// TIA Portal V16 program export: 1 tag tables, 6 data types, 52 data blocks, 60 code blocks (in call order from the OBs), 9 instance data blocks

VAR_GLOBAL   // PLC tag table "Default tag table"
   "E0.4" AT %I0.4 : Bool;   // CONTROLLO SALDATORE FILM
   "E0.5" AT %I0.5 : Bool;   // RICHIESTA APERTURA PORTA
   "E0.6" AT %I0.6 : Bool;   // PRESSOSTATO MACCHINA
   "E0.7" AT %I0.7 : Bool;   // ALLARME TERMICO MACCHINA
   "E1.0" AT %I1.0 : Bool;   // EMERGENZA MACCHINA
   "E1.1" AT %I1.1 : Bool;   // BARRIERE IMPEGNATE ENTRATA
   "E1.2" AT %I1.2 : Bool;   // BARRIERE IMPEGNATE USCITA
   "E1.3" AT %I1.3 : Bool;   // RESET MACCHINA
   "E1.4" AT %I1.4 : Bool;   // MARCIA AUTOMATICA MACCHINA
   "E1.5" AT %I1.5 : Bool;   // ARRESTO MACCHINA
   "E2.0" AT %I2.0 : Bool;   // TAVOLA IN FASE
   "E2.1" AT %I2.1 : Bool;   // [spare] COMANDO FRENO MOTORE ROTAZIONE
   "E2.2" AT %I2.2 : Bool;   // CARRELLO BASSO
   "E2.3" AT %I2.3 : Bool;   // CARRELLO ALTO
   "E2.4" AT %I2.4 : Bool;   // TAGLIO INDIETRO
   "E2.5" AT %I2.5 : Bool;   // TAGLIO AVANTI
   "E2.6" AT %I2.6 : Bool;   // CONTRASTO SALDATORE INDIETRO
   "E2.7" AT %I2.7 : Bool;   // CONTRASTO SALDATORE BASSO
   "E3.0" AT %I3.0 : Bool;   // RISERVA
   "E3.1" AT %I3.1 : Bool;   // RISERVA
   "E3.2" AT %I3.2 : Bool;   // LETTURA CENTRAGGIO PALLET TRASPORTO CENTRO MACCHINA
   "E3.3" AT %I3.3 : Bool;   // CONTEGGIO CENTRAGGIO PALLET TRASPORTO CENTRO MACCHINA
   "E3.4" AT %I3.4 : Bool;   // CONTROLLO ROTAZIONE TAVOLA IN ENTRATA E LETTURA LUNGHEZZA PALLET
   "E3.5" AT %I3.5 : Bool;   // CONTROLLO ROTAZIONE TAVOLA IN USCITA E FINE CICLO
   "E3.6" AT %I3.6 : Bool;   // SEGNALE PALLET PRONTO IN ENTRATA
   "E3.7" AT %I3.7 : Bool;   // SEGNALE PRONTO A RICEVERE IN USCITA
   "E4.0" AT %I4.0 : Bool;   // SEGNALE FINE TRASFERIMENTO PALLET IN USCITA
   "E4.1" AT %I4.1 : Bool;   // SEGNALE ESCLUSIONE FASCIATURA
   "E4.2" AT %I4.2 : Bool;   // POSIZIONAMENTO PALLET TRASPORTO POS. 01
   "E4.3" AT %I4.3 : Bool;   // POSIZIONAMENTO PALLET TRASPORTO POS. 02
   "E4.4" AT %I4.4 : Bool;   // POSIZIONAMENTO PALLET TRASPORTO POS. 03
   "E4.5" AT %I4.5 : Bool;   // POSIZIONAMENTO PALLET TRASPORTO POS. 04
   "E4.6" AT %I4.6 : Bool;   // POSIZIONAMENTO PALLET TRASPORTO POS. 05
   "E5.1" AT %I5.1 : Bool;   // POSIZIONAMENTO PALLET TRASPORTO POS. 08
   "E5.3" AT %I5.3 : Bool;   // [B2783] CONTROLLO 2 POSIZIONAMENTO POS. 05
   "E6.0" AT %I6.0 : Bool;   // CARRELLO BASSO (TOP)
   "E6.1" AT %I6.1 : Bool;   // CARRELLO ALTO (TOP)
   "E6.2" AT %I6.2 : Bool;   // LETTURA ALTEZZA PALLET (TOP)
   "E6.3" AT %I6.3 : Bool;   // PINZA CHIUSA BLOCCO FILM (TOP)
   "E6.4" AT %I6.4 : Bool;   // TAGLIO FILM AVANTI (TOP)
   "E6.5" AT %I6.5 : Bool;   // TAGLIO FILM INDIETRO (TOP)
   "E6.6" AT %I6.6 : Bool;   // ROTTURA ESAURIMENTO FILM (TOP)
   "E7.0" AT %I7.0 : Bool;   // CARRELLO INDIETRO (TOP)
   "E7.1" AT %I7.1 : Bool;   // CARRELLO AVANTI POSIZIONE TAGLIO (TOP)
   "E7.3" AT %I7.3 : Bool;   // PINZA CHIUSA TRAINO FILM (TOP)
   "E7.4" AT %I7.4 : Bool;   // SICUREZZA AVANZAMENTO (TOP)
   "E7.5" AT %I7.5 : Bool;   // SICUREZZA DISCESA (TOP) SX
   "E7.6" AT %I7.6 : Bool;   // SICUREZZA DISCESA (TOP) DX
   "E7.7" AT %I7.7 : Bool;   // SICUREZZA CONTROLLO SGANCIO FRENI SAL.-DISC. (TOP)
   HSC2Value AT %ID1004 : DInt;   // Counter value for HSC2
   HSC1Value AT %ID1000 : DInt;
   "E4.7" AT %I4.7 : Bool;   // POSIZIONAMENTO PALLET TRASPORTO POS. 06
   "E5.0" AT %I5.0 : Bool;   // POSIZIONAMENTO PALLET TRASPORTO POS. 07
   "E5.2" AT %I5.2 : Bool;   // [B2782] CONTROLLO 1 POSIZIONAMENTO POS. 05
   "E5.4" AT %I5.4 : Bool;   // SEGNALE PORTA TAGLIAFUOCO APERTA
   "E5.5" AT %I5.5 : Bool;   // SEGNALE CHIUSURA PORTA TAGLIAFUOCO
   "E5.6" AT %I5.6 : Bool;   // SelectorBypass
   "E5.7" AT %I5.7 : Bool;   // Free
   "E6.7" AT %I6.7 : Bool;   // SPARE - NOT USED
   "E7.2" AT %I7.2 : Bool;   // RISERVA
   "A0.0" AT %Q0.0 : Bool;   // APERTURA PORTA
   "A0.1" AT %Q0.1 : Bool;   // EMERGENZA PLC SU PILZ
   "A0.2" AT %Q0.2 : Bool;   // EMERGENZA MACCHINA
   "A0.3" AT %Q0.3 : Bool;   // MARCIA AUTOMATICA MACCHINA
   "A0.4" AT %Q0.4 : Bool;   // SEGNALATORE ACUSTICO MARCIA
   "A0.6" AT %Q0.6 : Bool;   // FRENO MOTORE ROTAZIONE
   "A0.7" AT %Q0.7 : Bool;   // MOTORE ROTAZIONE
   "A1.0" AT %Q1.0 : Bool;   // FASCIA STRETTA
   "A1.1" AT %Q1.1 : Bool;   // CORDA STRETTA
   "A2.0" AT %Q2.0 : Bool;   // PINZA APERTA
   "A2.1" AT %Q2.1 : Bool;   // PINZA CHIUSA
   "A2.2" AT %Q2.2 : Bool;   // TAGLIO AVANTI / INDIETRO
   "A2.3" AT %Q2.3 : Bool;   // SOFFIO ARIA PER CODA FILM
   "A2.4" AT %Q2.4 : Bool;   // TAGLIO FILM
   "A2.5" AT %Q2.5 : Bool;   // SALDATORE FILM
   "A2.6" AT %Q2.6 : Bool;   // CONTRASTO SALDATORE AVANTI
   "A2.7" AT %Q2.7 : Bool;   // CONTRASTO SALDATORE INDIETRO
   "A3.0" AT %Q3.0 : Bool;   // CONTRASTO SALDATORE SALITA/DISCESA
   "A3.1" AT %Q3.1 : Bool;   // RISERVA
   "A3.2" AT %Q3.2 : Bool;   // RISERVA
   "A3.3" AT %Q3.3 : Bool;   // MOTORE TRASPORTO CENTRO MACCHINA
   "A3.4" AT %Q3.4 : Bool;   // SEGNALE PRONTO A RICEVERE IN ENTRATA
   "A3.5" AT %Q3.5 : Bool;   // SEGNALE FINE TRASFERIMENTO PALLET IN ENTRATA
   "A3.6" AT %Q3.6 : Bool;   // SEGNALE PALLET PRONTO IN USCITA
   "A3.7" AT %Q3.7 : Bool;   // SEGNALE PRONTO PER CHIUSURA PORTA TAGLIAFUOCO
   "A4.0" AT %Q4.0 : Bool;   // MOTORE TRASPORTO POS. 01 AVANTI
   "A4.1" AT %Q4.1 : Bool;   // MOTORE TRASPORTO POS. 02 AVANTI
   "A4.2" AT %Q4.2 : Bool;   // MOTORE TRASPORTO POS. 03 AVANTI
   "A4.3" AT %Q4.3 : Bool;   // MOTORE TRASPORTO POS. 04 AVANTI
   "A4.4" AT %Q4.4 : Bool;   // MOTORE TRASPORTO POS. 05 AVANTI
   "A4.5" AT %Q4.5 : Bool;   // MOTORE TRASPORTO POS. 06 AVANTI
   "A4.6" AT %Q4.6 : Bool;   // MOTORE TRASPORTO POS. 07 AVANTI
   "A4.7" AT %Q4.7 : Bool;   // MOTORE TRASPORTO POS. 08 AVANTI
   "A5.0" AT %Q5.0 : Bool;   // Lamp By-pass
   Motor_Tapete_Centrador AT %Q5.1 : Bool;   // SPARE - NOT USED
   Motor_Centrador_Sentido_Direto AT %Q5.2 : Bool;   // SPARE - NOT USED
   Motor_Centrador_Sentido_Inverso AT %Q5.3 : Bool;   // SPARE - NOT USED
   "A6.0" AT %Q6.0 : Bool;   // MOTORE CARRELLO (TOP) AVANTI
   "A6.1" AT %Q6.1 : Bool;   // MOTORE CARRELLO (TOP) INDIETRO
   "A6.2" AT %Q6.2 : Bool;   // START INVERTER SALITA CARRELLO (TOP)
   "A6.3" AT %Q6.3 : Bool;   // START INVERTER DISCESA CARRELLO (TOP)
   "A6.4" AT %Q6.4 : Bool;   // FRENO MOTORE (TOP) SALITA/DISCESA
   "A6.5" AT %Q6.5 : Bool;   // PINZA APERTA BLOCCO FILM (TOP)
   "A6.6" AT %Q6.6 : Bool;   // PINZA CHIUSA BLOCCO FILM (TOP)
   "A6.7" AT %Q6.7 : Bool;   // TAGLIO FILM AVANTI (TOP)
   "A7.0" AT %Q7.0 : Bool;   // TAGLIO FILM INDIETRO (TOP)
   "A7.1" AT %Q7.1 : Bool;   // PINZA APERTA TRAINO FILM (TOP)
   "A7.2" AT %Q7.2 : Bool;   // PINZA CHIUSA TRAINO FILM (TOP)
   "A5.4" AT %Q5.4 : Bool;   // SPARE - NOT USED
   "A5.5" AT %Q5.5 : Bool;   // SPARE - NOT USED
   "A5.6" AT %Q5.6 : Bool;   // SPARE - NOT USED
   "A0.5" AT %Q0.5 : Bool;   // ENABLE INVERTER ROTAZIONE
   "A5.7" AT %Q5.7 : Bool;   // SPARE - NOT USED
   "A10.0" AT %Q10.0 : Bool;   // SPARE - NOT USED
   "A10.1" AT %Q10.1 : Bool;   // SPARE - NOT USED
   "A10.2" AT %Q10.2 : Bool;   // SPARE - NOT USED
   "A10.3" AT %Q10.3 : Bool;   // SPARE - NOT USED
   "A7.3" AT %Q7.3 : Bool;   // SPARE - NOT USED
   "A7.4" AT %Q7.4 : Bool;   // SPARE - NOT USED
   "A7.5" AT %Q7.5 : Bool;   // SPARE - NOT USED
   "A7.6" AT %Q7.6 : Bool;   // SPARE - NOT USED
   "A7.7" AT %Q7.7 : Bool;   // SPARE - NOT USED
   "M0.0" AT %M0.0 : Bool;   // Machine cycle: M0.0 Start cycle
   "M0.1" AT %M0.1 : Bool;   // Machine cycle: M0.1 Waiting for top before
   "M0.2" AT %M0.2 : Bool;   // Machine cycle: M0.2 Loading data for spool carriage position
   "M0.3" AT %M0.3 : Bool;   // Machine cycle: M0.3 Waiting for pressure plate and lifter
   "M0.4" AT %M0.4 : Bool;   // Machine cycle: M0.4 Spool carriage upward/downward with rotation
   "M0.5" AT %M0.5 : Bool;   // Machine cycle: M0.5 Table rotation - Table revolution counter
   "M0.6" AT %M0.6 : Bool;   // Machine cycle: M0.6 Load new data for next spool carriage height
   "M0.7" AT %M0.7 : Bool;   // Machine cycle: M0.7 Spool carriage upward/downward with rotation
   "M1.0" AT %M1.0 : Bool;   // Machine cycle: M1.0 Revolution over welder contrast
   "M1.1" AT %M1.1 : Bool;   // Machine cycle: M1.1
   "M1.2" AT %M1.2 : Bool;   // Machine cycle: M1.2 Table rotation deceleration
   "M1.3" AT %M1.3 : Bool;   // Machine cycle: M1.3 Table rotation deceleration
   "M1.4" AT %M1.4 : Bool;   // Machine cycle: M1.4 Stop table rotation - Waiting step
   "M1.5" AT %M1.5 : Bool;   // Machine cycle: M1.5 Waiting step
   "M1.6" AT %M1.6 : Bool;   // Machine cycle: M1.6 Pallet unload
   "M1.7" AT %M1.7 : Bool;   // Machine cycle: M1.7 Clamp and top check
   "M2.0" AT %M2.0 : Bool;   // Machine cycle: V2.0 Label cycle 1st label
   "M2.2" AT %M2.2 : Bool;   // Machine cycle: M2.2 Clamp and top check (Test cycle)
   "M2.3" AT %M2.3 : Bool;   // Machine cycle: M2.3 Checking step (Test cycle)
   "M2.4" AT %M2.4 : Bool;   // Label cycle
   "M3.0" AT %M3.0 : Bool;   // Machine cycle: M3.0 Table rotation middle speed
   "M3.1" AT %M3.1 : Bool;   // Machine cycle: M3.1 Table rotation deceleration
   "M3.2" AT %M3.2 : Bool;   // Machine cycle: M3.2 Table rotation deceleration
   "M3.3" AT %M3.3 : Bool;   // Machine cycle: M3.3 Waiting for top cycle
   "M5.0" AT %M5.0 : Bool;   // Top cycle: V5.0 Start cycle
   "M5.1" AT %M5.1 : Bool;   // Top cycle: V5.1 Closing clamp to pull top film
   "M5.2" AT %M5.2 : Bool;   // Top cycle: V5.2 Opening clamp to block top film
   "M5.3" AT %M5.3 : Bool;   // Top cycle: V5.3 Top carriage forward
   "M5.4" AT %M5.4 : Bool;   // Top cycle: V5.4 Closing clamp to block top film
   "M5.5" AT %M5.5 : Bool;   // Top cycle: V5.5 Top carriage down
   "M5.6" AT %M5.6 : Bool;   // Top cycle: V5.6 Top carriage on pallet top
   "M5.7" AT %M5.7 : Bool;   // Top cycle: V5.7 Top cutter forward
   "M6.0" AT %M6.0 : Bool;   // Top cycle: V6.0 Top cutter backward
   "M6.1" AT %M6.1 : Bool;   // Top cycle: V6.1 Top carriage forward\Top cutter backward
   "M6.2" AT %M6.2 : Bool;   // Top cycle: V6.2 Top carriage downward to pull down top film
   "M6.3" AT %M6.3 : Bool;   // Top cycle: V6.3 Top carriage downward to release top film
   "M6.4" AT %M6.4 : Bool;   // Top cycle: V6.4 Top carriage stopped against vibration
   "M6.5" AT %M6.5 : Bool;   // Top cycle: V6.5 Top carriage upward
   "M6.6" AT %M6.6 : Bool;   // Top cycle: V6.6 Top carriage upward and backward
   "M6.7" AT %M6.7 : Bool;   // Top cycle: V6.7 Waiting for Rotoplat end cycle
   "M8.0" AT %M8.0 : Bool;   // Top film ended cycle: V8.0 Top carriage backward
   "M8.1" AT %M8.1 : Bool;   // Top film ended cycle: V8.1 Top carriage downward
   "M8.2" AT %M8.2 : Bool;   // Top film ended cycle: V8.2 Top carriage forward
   "M8.3" AT %M8.3 : Bool;   // Top film ended cycle: V8.3 Wait for reset button
   "M8.4" AT %M8.4 : Bool;   // Top film ended cycle: V8.4 Wait for automatic mode
   "M8.5" AT %M8.5 : Bool;   // Top film ended cycle: V8.5 Top carriage backward
   "M8.6" AT %M8.6 : Bool;   // Top film ended cycle: V8.6 Top carriage upward
   "M9.0" AT %M9.0 : Bool;   // Top cycle: V9.0 Top carriage downward for 90 degree top
   "M9.1" AT %M9.1 : Bool;   // Top cycle: V9.1 Wait step 1 for 90 degree top
   "M9.2" AT %M9.2 : Bool;   // Top cycle: V9.2 Top carriage upward for 90 degree top
   "M9.3" AT %M9.3 : Bool;   // Top cycle: V9.3 Wait step 2 for 90 degree top
   "M9.4" AT %M9.4 : Bool;   // Top cycle: V9.4 Waiting step 3 for 90 degree top after top
   "M9.5" AT %M9.5 : Bool;   // Top cycle: V9.5 Top carriage upward for 90 degree top
   "M9.6" AT %M9.6 : Bool;   // Top cycle: V9.6 Wait step 4 for 90 degree top after top
   Alarm AT %M10.0 : Bool;   // Main emergency
   "M10.1" AT %M10.1 : Bool;   // Prearrangement automatic cycle
   Manu AT %M10.2 : Bool;   // Manual mode
   Auto AT %M10.3 : Bool;   // Automatic mode
   "M10.4" AT %M10.4 : Bool;   // Automatic mode for film ended or broken
   Stop AT %M10.5 : Bool;   // Memory stop cycle
   "M10.6" AT %M10.6 : Bool;   // Memory to stop cycle for door open request
   Warning AT %M10.7 : Bool;   // Warning message active
   "M11.5" AT %M11.5 : Bool;   // Button Reset support memory
   "M11.6" AT %M11.6 : Bool;   // Memory release Button Reset
   FilmEnd AT %M12.0 : Bool;   // Film ended or broken
   TopEnd AT %M12.1 : Bool;   // Top film ended or broken
   On AT %M12.7 : Bool;   // Bit always on
   "M14.7" AT %M14.7 : Bool;   // Table rotation backward to reset encoder
   Reset AT %M15.0 : Bool;   // Main reset
   "M15.1" AT %M15.1 : Bool;   // Request to reset spool carriage encoder
   "M15.2" AT %M15.2 : Bool;   // First cycle
   TransitIn AT %M15.3 : Bool;   // Pallet transit in infeed
   TransitOut AT %M15.4 : Bool;   // Pallet transit in outfeed
   TransitInBkw AT %M15.5 : Bool;   // Transit memory in infeed from reverse
   V15_6 AT %M15.6 : Bool;   // Automatic mode for external conveyors
   "M15.7" AT %M15.7 : Bool;   // Request to reset table rotation encoder
   "M16.0" AT %M16.0 : Bool;   // Conveyor cycle: M16.0 Start cycle
   "M16.1" AT %M16.1 : Bool;   // Conveyor cycle: M16.1 Loading pallet
   "M16.2" AT %M16.2 : Bool;   // Conveyor cycle: M16.2 Pallet positioned
   "M16.3" AT %M16.3 : Bool;   // Conveyor cycle: M16.3 Unloading pallet
   "M16.4" AT %M16.4 : Bool;   // Conveyor cycle: M16.4 Loading/unloading pallet simultaneously
   "M16.5" AT %M16.5 : Bool;   // Conveyor cycle: M16.5 Unloading pallet
   "M16.6" AT %M16.6 : Bool;   // Conveyor cycle: M16.6 Loading pallet from reverse
   "M16.7" AT %M16.7 : Bool;   // Conveyor cycle: M16.7 Pallet positioned from reverse
   "M17.0" AT %M17.0 : Bool;   // Pallet load cycle: V17.0 Table rotation to load phase
   "M17.1" AT %M17.1 : Bool;   // Pallet load cycle: V17.1 Table rotation to machine phase from load
   "M17.2" AT %M17.2 : Bool;   // Pallet load cycle: V17.2 Table rotation to unload phase
   "M17.3" AT %M17.3 : Bool;   // Pallet load cycle: V17.3 Table rotation to machine phase from unload
   "M17.4" AT %M17.4 : Bool;   // Pallet load cycle: V17.4 Table rotation to reverse phase
   "M17.5" AT %M17.5 : Bool;   // Pallet load cycle: V17.5 Table rotation to machine phase from re
   "M18.0" AT %M18.0 : Bool;   // Ring clamp cycle: M18.0 Start cycle
   "M18.1" AT %M18.1 : Bool;   // Ring clamp cycle: M18.1 Open clamp
   "M18.2" AT %M18.2 : Bool;   // Ring clamp cycle: M18.2 Waiting for welder contrast up
   "M18.3" AT %M18.3 : Bool;   // Ring clamp cycle: M18.3 Waiting table deceleration
   "M18.4" AT %M18.4 : Bool;   // Ring clamp cycle: M18.4 Ring clamp upward
   "M18.5" AT %M18.5 : Bool;   // Ring clamp cycle: M18.5 Opening ring clamp
   "M18.6" AT %M18.6 : Bool;   // Ring clamp cycle: M18.6 Waiting for table rotation in phase
   "M18.7" AT %M18.7 : Bool;   // Ring clamp cycle: M18.7 Closing ring clamp
   "M19.0" AT %M19.0 : Bool;   // Ring clamp cycle: M19.0 Welder and cut unit upward
   "M19.1" AT %M19.1 : Bool;   // Ring clamp cycle: M19.1 Waiting for welding time
   "M19.2" AT %M19.2 : Bool;   // Ring clamp cycle: M19.2 Welder unit downward
   "M19.3" AT %M19.3 : Bool;   // Ring clamp cycle: M19.3 Waiting for pallet unload
   "M20.0" AT %M20.0 : Bool;   // Claw clamp HS40 cycle: M20.0 Start cycle
   "M20.1" AT %M20.1 : Bool;   // Claw clamp HS40 cycle: M20.1 Opening clamp
   "M20.2" AT %M20.2 : Bool;   // Claw clamp HS40 cycle: M20.2 Waiting for table rotation in phase
   "M20.3" AT %M20.3 : Bool;   // Claw clamp HS40 cycle: M20.3 Closing clamp
   "M20.4" AT %M20.4 : Bool;   // Claw clamp HS40 cycle: M20.4 Welder and cut unit forward
   "M20.5" AT %M20.5 : Bool;   // Claw clamp HS40 cycle: M20.5 Waiting for cut and welding time
   "M20.6" AT %M20.6 : Bool;   // Claw clamp HS40 cycle: M20.6 Welder and cut unit backward
   "M22.0" AT %M22.0 : Bool;   // Spring clamp cycle: M22.0 Start cycle
   "M22.1" AT %M22.1 : Bool;   // Spring clamp cycle: M22.1 Open clamp
   "M22.2" AT %M22.2 : Bool;   // Spring clamp cycle: M22.2 Waiting for welder contrast up
   "M22.3" AT %M22.3 : Bool;   // Spring clamp cycle: M22.3 Waiting table deceleration
   "M22.4" AT %M22.4 : Bool;   // Spring clamp cycle: M22.4 Spring clamp upward
   "M22.5" AT %M22.5 : Bool;   // Spring clamp cycle: M22.5 Opening spring clamp
   "M22.6" AT %M22.6 : Bool;   // Spring clamp cycle: M22.6 Waiting for table rotation in phase
   "M22.7" AT %M22.7 : Bool;   // Spring clamp cycle: M22.7 Table rotation forward for twist
   "M23.0" AT %M23.0 : Bool;   // Spring clamp cycle: M23.0 Closing spring clamp
   "M23.1" AT %M23.1 : Bool;   // Spring clamp cycle: M23.1 Welder and cut unit upward
   "M23.2" AT %M23.2 : Bool;   // Spring clamp cycle: M23.2 Waiting for welding time
   "M23.3" AT %M23.3 : Bool;   // Spring clamp cycle: M23.3 Welder unit downward
   "M23.4" AT %M23.4 : Bool;   // Spring clamp cycle: M23.4 Waiting for welder contrast down
   "M30.0" AT %M30.0 : Bool;   // Film broken cycle: M30.0 Start cycle
   "M30.1" AT %M30.1 : Bool;   // Film broken cycle: M30.1 All unit to home position
   "M30.2" AT %M30.2 : Bool;   // Film broken cycle: M30.2 Spool carriage to film change position
   "M30.3" AT %M30.3 : Bool;   // Film broken cycle: M30.3 Waiting for alarm mode
   "M30.4" AT %M30.4 : Bool;   // Film broken cycle: M30.4 Waiting automatic mode
   "M30.5" AT %M30.5 : Bool;   // Film broken cycle: M30.5 Spool carriage downward
   "M30.6" AT %M30.6 : Bool;   // Film broken cycle: M30.6 Waiting step
   "M32.0" AT %M32.0 : Bool;   // Film broken cycle 1: M32.0 Start cycle
   "M32.1" AT %M32.1 : Bool;   // Film broken cycle 1: M32.1 Table rotation middle speed
   "M32.2" AT %M32.2 : Bool;   // Film broken cycle 1: M32.2 Table rotation middle speed
   "M32.3" AT %M32.3 : Bool;   // Film broken cycle 1: M32.3 Table rotation deceleration
   "M32.4" AT %M32.4 : Bool;   // Film broken cycle 1: M32.4 Table rotation deceleration
   "M32.5" AT %M32.5 : Bool;   // Film broken cycle 1: M32.5 Waiting step
   V50_1 AT %M50.1 : Bool;   // Infeed conveyor pos.1 load
   V50_6 AT %M50.6 : Bool;   // Transit memory pos6->pos7
   V51_1 AT %M51.1 : Bool;   // Memory to exclude wrapping in pos 1
   V56_0 AT %M56.0 : Bool;   // Start cycle lifter pos.2: V56.0 Lifter empty and low
   V56_1 AT %M56.1 : Bool;   // Start cycle lifter pos.2: V56.1 Lifter upstroke
   V56_2 AT %M56.2 : Bool;   // Start cycle lifter pos.2: V56.2 Waiting step - pallet load
   V56_3 AT %M56.3 : Bool;   // Start cycle lifter pos.2: V56.3 Lifter downstroke
   V56_4 AT %M56.4 : Bool;   // Start cycle lifter pos.2: V56.4 Waiting step - pallet unload
   V56_5 AT %M56.5 : Bool;   // Start cycle lifter pos.2: V56.5
   V56_6 AT %M56.6 : Bool;   // Start cycle lifter pos.2: V56.6
   V57_0 AT %M57.0 : Bool;   // Load to pos1 with forklift request
   V57_1 AT %M57.1 : Bool;   // Load to pos1 with forklift ok
   V57_2 AT %M57.2 : Bool;   // Unload from pos1 with forklift request
   V57_3 AT %M57.3 : Bool;   // Unload from pos1 with forklift OK
   V57_5 AT %M57.5 : Bool;   // Start cycle pos.1 OK
   Sgn_TopPosizTransfer AT %M64.1 : Bool;   // Top Out Supp. Out - Signal " Top In Position for Pallet Transfe
   ContrastCarriageOk1 AT %M70.0 : Bool;   // ContrastCarriageOK1: Contrast carriage in position to return to start cycle
   ContrastCarriageOk4 AT %M70.3 : Bool;   // ContrastCarriageOk4: Contrast carriage in position for film broken cycle
   ContrastCarriageOk7 AT %M70.6 : Bool;   // ContrastCarriageOk7: Contrast carriage unit in position to begin cycle
   ContrastCarriageOk17 AT %M72.0 : Bool;   // ContrastCarriageOk17: Contrast carriage in position for pallet transit
   ClampCutOk1 AT %M80.0 : Bool;   // ClampCutOK1: Clamp and cutter in position to return to start cycle
   ClampCutOk2 AT %M80.1 : Bool;   // ClampCutOK2: Film tail wrapped
   ClampCutOk3 AT %M80.2 : Bool;   // ClampCutOK3: Main emergency (1+) for welder circuit control
   ClampCutOk4 AT %M80.3 : Bool;   // ClampCutOk4: Clamp in position for film broken cycle
   ClampCutOk5 AT %M80.4 : Bool;   // ClampCutOk5: Revolution over welder contrast done
   ClampCutOk6 AT %M80.5 : Bool;   // ClampCutOk6: Clamp and cutter cycle ended
   ClampCutOk7 AT %M80.6 : Bool;   // ClampCutOk7: Clamp and cutter units in position to begin cycle
   ClampCutOk8 AT %M80.7 : Bool;   // ClampCutOk8: Table rotation middle speed
   ClampCutOk9 AT %M81.0 : Bool;
   ClampCutOk10 AT %M81.1 : Bool;   // ClampCutOk10: Clamp and cut unit in safety position for table rotation
   ClampCutOK11 AT %M81.2 : Bool;   // ClampCutOk11: Exclude deceleration not correct alarm
   ClampCutOK12 AT %M81.3 : Bool;   // ClampCutOk12: Film request during clamp cycle
   ClampCutOk13 AT %M81.4 : Bool;   // ClampCutOk13: Request to move spool carrage up at the begining
   ClampCutOk14 AT %M81.5 : Bool;   // ClampCutOk14: Ok to move spool carrage down at the begining
   ClampCutOk15 AT %M81.6 : Bool;   // ClampCutOk15: Request to move spool carrage up to cover film tail
   ClampCutOk16 AT %M81.7 : Bool;   // ClampCutOk16: Ok to move spool carrage down to cover film tail
   ClampCutOk17 AT %M82.0 : Bool;   // ClampCutOk17: Clamp units in position for pallet transit
   ClampCutOk18 AT %M82.1 : Bool;   // ClampCutOk18: Enable for spool carriage downward at cycle end
   ClampCutOk19 AT %M82.2 : Bool;   // ClampCutOk19: Clamp and cut unit in safety position for pallet lifter
   ClampCutOk20 AT %M82.3 : Bool;   // Pallet backward request for ClampCut cycle
   ClampCutOk21 AT %M82.4 : Bool;   // ClampCutOk21: Cutter arm forward
   "M83.0" AT %M83.0 : Bool;   // Table rotation forward for twist
   "M83.1" AT %M83.1 : Bool;   // Table rotation backward for twist
   LifterOK1 AT %M84.0 : Bool;   // LifterOK1: Pallet lifter down
   LifterOk2 AT %M84.1 : Bool;   // LifterOk2: Pallet lifter up
   "M84.3" AT %M84.3 : Bool;   // Pallet lifter upward
   "M84.4" AT %M84.4 : Bool;   // Pallet lifter downward
   RopeUnitOk1 AT %M84.5 : Bool;   // RopeUnitOk1: Rope unit open
   RopeUnitOk2 AT %M84.6 : Bool;   // RopeUnitOk2: Full rope unit open
   TopOK1 AT %M85.0 : Bool;   // Top carriage OK1: Top cycle ended
   TopOK2 AT %M85.1 : Bool;   // Top carriage OK2: Ok for pressure plate downward on 90 degree top
   TopOK3 AT %M85.2 : Bool;   // Top carriage OK3: Top carriage backward or forward
   TopOk4 AT %M85.3 : Bool;   // Top carriage OK4: Top carriage up
   TopOk5 AT %M85.6 : Bool;   // Top carriage OK5: Top cycle ended for top dustproof
   TopOk6 AT %M85.7 : Bool;   // Top carriage OK6: Emergency rele' on pilz chain
   PressureOk1 AT %M86.0 : Bool;   // PressureOk1: Pressure plate on pallet
   PressureOk2 AT %M86.1 : Bool;   // PressureOk2: Pressure plate up
   PressureOk3 AT %M86.2 : Bool;   // PressureOk3: Pressure plate Ok for pallet height
   "M86.3" AT %M86.3 : Bool;   // Pressure plate downward
   "M86.4" AT %M86.4 : Bool;   // Pressure plate upward
   V86_5 AT %M86.5 : Bool;   // Pressure Plate downstroke request
   V87_0 AT %M87.0 : Bool;   // Top carriage forward
   V87_1 AT %M87.1 : Bool;   // Top carriage backward
   V87_2 AT %M87.2 : Bool;   // Top carriage forward/backward slow speed
   V87_3 AT %M87.3 : Bool;   // Table rotation forward for top
   V87_4 AT %M87.4 : Bool;   // Table rotation backward for top
   TopOk7 AT %M88.0 : Bool;   // TopOk7: Top carriage backward
   TopOk8 AT %M88.1 : Bool;   // TopOK8: All top units in position for automatic cycle
   TopOk9 AT %M88.2 : Bool;   // TopOk3: Top before cycle ended
   TopOk10 AT %M88.4 : Bool;   // TopOk10: Table rotation middle speed
   TopOk11 AT %M88.5 : Bool;   // Top carriage OK11: All top units OK for automatic cycle
   TopOk12 AT %M88.6 : Bool;   // Top carriage OK12: Carriage downward for top 90 ended cycle
   V89_0 AT %M89.0 : Bool;   // Table rotation for top cycle (Top->Table)
   V89_1 AT %M89.1 : Bool;   // Fast speed table rotation for top cycle (Top->Table)
   V89_2 AT %M89.2 : Bool;   // Middle speed table rotation for top cycle (Top->Table)
   V89_3 AT %M89.3 : Bool;   // Spool carriage downward for top cycle (Top->Table)
   V89_4 AT %M89.4 : Bool;   // Spool carriage upward for top cycle (Top->Table)
   V89_5 AT %M89.5 : Bool;   // Memory to control the top cycle reset (Top->Table)
   Top_OFF AT %M89.6 : Bool;   // Top off by the machine configuration
   Top_ON AT %M89.7 : Bool;   // Top on by the machine configuration
   ConvOk1 AT %M90.0 : Bool;   // ConvOk1: Pallet ready to be wrapped
   ConvOk2 AT %M90.1 : Bool;   // ConvOk2: Pallet in position to return to start cycle
   ConvOk3 AT %M90.2 : Bool;   // ConvOk3: Conveyor is running
   ConvOk4 AT %M90.3 : Bool;   // ConvOk4: Forward for inverter
   ConvOk5 AT %M90.4 : Bool;   // ConvOK5: Fast speed for conveyor
   ConvOk6 AT %M90.5 : Bool;   // ConvOk6: Slow speed for conveyor
   ConvOk7 AT %M90.6 : Bool;   // ConvOk7: Backward for inverter
   V90_7 AT %M90.7 : Bool;   // ConvOk8: Conveyor is running
   "M91.0" AT %M91.0 : Bool;   // Load data from table to display
   "M91.1" AT %M91.1 : Bool;   // Load data from display to table
   "M91.2" AT %M91.2 : Bool;   // Program active is Ok
   TechnoplatOk1 AT %M92.0 : Bool;   // TechnoplatOk1: All unit to home position
   TechnoplatOk2 AT %M92.1 : Bool;   // TechnoplatOk2: Reset all cycle
   TechnoplatOk3 AT %M92.2 : Bool;   // TechnoplatOk3: A manual operation has been done
   TechnoplatOk4 AT %M92.3 : Bool;   // TechnoplatOk4: Top unit is able to start his cycle
   TechnoplatOk5 AT %M92.4 : Bool;   // TechnoplatOk5:
   TechnoplatOk6 AT %M92.5 : Bool;   // TechnoplatOk6:
   "M93.0" AT %M93.0 : Bool;   // One shot rising (OSR) for table phase sensor
   "M93.1" AT %M93.1 : Bool;   // One shot falliing (OSF) for table phase sensor
   StopRequest AT %M93.5 : Bool;   // (Memory) Stop request by operator button
   V94_0 AT %M94.0 : Bool;   // Spool carriage upward request for table cycle
   V94_1 AT %M94.1 : Bool;   // Spool carriage downward request for table cycle
   E01 AT %M100.0 : Bool;   // Spool carriage encoder channel A (Technoplat)
   E02 AT %M100.1 : Bool;   // Spool carriage encoder channel B (Technoplat)
   E03_NotUsed AT %M100.2 : Bool;   // Safety barriers excluded by selector (Barrier)
   E04 AT %M100.3 : Bool;   // Infeed safety barrier engaged (Barrier)
   E05 AT %M100.4 : Bool;   // Outfeed safety barrier engaged (Barrier)
   E06 AT %M100.5 : Bool;   // Reset button (Technoplat)
   E07_NotUsed AT %M100.6 : Bool;   // Key selector automatic (0)/manual (1) mode (Technoplat)
   E08 AT %M100.7 : Bool;   // Automatic functioning button (Technoplat)
   E09 AT %M101.0 : Bool;   // Stop request by operator button (Technoplat)
   E10 AT %M101.1 : Bool;   // Request to open door key selector (1 open) (Technoplat)
   E11 AT %M101.2 : Bool;   // Pressure switch (Technoplat)
   E12 AT %M101.3 : Bool;   // Thermic alarm (Technoplat)
   E13 AT %M101.4 : Bool;   // Fault inverter (Technoplat)
   E14 AT %M101.5 : Bool;   // Emergency stop push button (Technoplat)
   E15 AT %M101.6 : Bool;   // Main emergency 1+ (Technoplat)
   E16 AT %M101.7 : Bool;   // Spool carriage down (Technoplat)
   E17 AT %M102.0 : Bool;   // Spool carriage up (Technoplat)
   E18 AT %M102.1 : Bool;   // Reading pallet height on spool carriage (Technoplat)
   E19 AT %M102.2 : Bool;   // Film broken or ended on spool carriage (Technoplat)
   E20 AT %M102.3 : Bool;   // Film at 10% on spool carriage (Technoplat)
   E21_NotUsed AT %M102.4 : Bool;   // Reading pallet height on spool carriage with reflector (Technoplat)
   E22 AT %M102.5 : Bool;   // Table rotation phase sensor (Technoplat)
   E23_NotUsed AT %M102.6 : Bool;   // Pallet lifter down (Lifter)
   E24 AT %M102.7 : Bool;   // Pressure plate up (Pressure plate)
   E25 AT %M103.0 : Bool;   // Single rope unit open (Rope unit)
   E26_NotUsed AT %M103.1 : Bool;   // Table rotation phase 2 sensor for top (Technoplat)
   E27_NotUsed AT %M103.2 : Bool;   // Upper(double) rope unit open (Rope unit)
   E28 AT %M103.3 : Bool;   // Pressure plate positioning
   E29 AT %M103.4 : Bool;   // Table rotation load phase sensor (Technoplat)
   E30 AT %M103.5 : Bool;   // Table rotation unload phase sensor (Technoplat)
   E31 AT %M103.6 : Bool;   // Lower (double) rope unit closed (Rope unit)
   E32 AT %M103.7 : Bool;
   E33 AT %M104.0 : Bool;   // Scanner start pushbutton (pos2)
   E34 AT %M104.1 : Bool;   // Labeler start pushbutton (pos3)
   E35 AT %M104.2 : Bool;   // SelectotBypass
   E36 AT %M104.3 : Bool;
   E37 AT %M104.4 : Bool;   // Infeed table rotation control (Conveyor)
   E38 AT %M104.5 : Bool;   // Pallet position control in infeed (Conveyor)
   E39 AT %M104.6 : Bool;   // Pallet position control in outfeed (Conveyor)
   E40 AT %M104.7 : Bool;   // Outfeed table rotation control-End of cycle (Conveyor)
   E41 AT %M105.0 : Bool;   // Pallet position forward (Conveyor)
   E42 AT %M105.1 : Bool;
   E43 AT %M105.2 : Bool;   // Pallet ready in infeed signal (Std signal)
   E44 AT %M105.3 : Bool;   // Ready to receive pallet from outfeed signal (Std signal)
   E45 AT %M105.4 : Bool;   // End of pallet transfer signal (Std signal)
   E46 AT %M105.5 : Bool;   // Wrapping excluded signal (Std signal)
   E47 AT %M105.6 : Bool;   // Pallet ready from reverse
   E48 AT %M105.7 : Bool;
   E49 AT %M106.0 : Bool;   // Wrapping excluded signal (Std signal)
   E50 AT %M106.1 : Bool;
   E51 AT %M106.2 : Bool;   // Signal 1 for program selection by external signal (Std Signal)
   E52 AT %M106.3 : Bool;   // Signal 2 for program selection by external signal (Std Signal)
   E53 AT %M106.4 : Bool;   // Signal 3 for program selection by external signal (Std Signal)
   E54 AT %M106.5 : Bool;   // Signal 4 for program selection by external signal (Std Signal)
   E55_NotUsed AT %M106.6 : Bool;   // Customer conveyor stopped signal (No conveyor signal)
   E56_NotUsed AT %M106.7 : Bool;   // Start wrapping signal (No conveyor signal)
   E57 AT %M107.0 : Bool;
   E58 AT %M107.1 : Bool;
   E59 AT %M107.2 : Bool;   // Coil for welder control (All clamp)
   E60 AT %M107.3 : Bool;   // Film clamp closed (RingSpring clamp)
   E61 AT %M107.4 : Bool;   // Film clamp open (Ring clamp)
   E62_NotUsed AT %M107.5 : Bool;   // Film clamp down (RingSpring clamp)
   E63_NotUsed AT %M107.6 : Bool;   // Film clamp up (Ring clamp)
   E64 AT %M107.7 : Bool;   // Welder contrast down (RingSpring clamp)
   E65 AT %M108.0 : Bool;   // Welder contrast back (Contrast carriage)
   E66 AT %M108.1 : Bool;   // Welder unit down (RingSpring clamp)
   E67 AT %M108.2 : Bool;   // Welder unit up (Ring clamp)
   E68 AT %M108.3 : Bool;   // Clamp carriage forward (Spring clamp)
   E69 AT %M108.4 : Bool;   // Clamp carriage backward (Spring clamp)
   E70 AT %M108.5 : Bool;   // Clamp carriage positioning (Spring clamp)
   E71 AT %M108.6 : Bool;   // Cutting and welding unit forward (Claw clamp)
   E72 AT %M108.7 : Bool;   // Cutting and welding unit backward (Claw clamp)
   E73 AT %M109.0 : Bool;   // Welder unit backward (Claw clamp)
   E74 AT %M109.1 : Bool;
   E75 AT %M109.2 : Bool;
   E76 AT %M109.3 : Bool;
   E77 AT %M109.4 : Bool;
   E78 AT %M109.5 : Bool;
   E79 AT %M109.6 : Bool;
   E80 AT %M109.7 : Bool;
   E81_NotUsed AT %M110.0 : Bool;   // Encoder (Robopac gear) for selfcenter system on preload sysyem (Conveyor)
   E82 AT %M110.1 : Bool;   // Encoder (Robopac gear) for selfcenter system (Conveyor)
   E83 AT %M110.2 : Bool;   // Deceleration for pallet position (Conveyor)
   E84 AT %M110.3 : Bool;   // Pallet positioning for selfcenter system (Conveyor)
   E85 AT %M110.4 : Bool;
   E86 AT %M110.5 : Bool;   // Infeed safety barrier photocell for muting by plc (Barrier)
   E87 AT %M110.6 : Bool;   // Outfeed safety barrier photocell for muting by plc (Barrier)
   E88 AT %M110.7 : Bool;
   E89 AT %M111.0 : Bool;
   E90 AT %M111.1 : Bool;
   E91 AT %M111.2 : Bool;
   E92 AT %M111.3 : Bool;
   E93 AT %M111.4 : Bool;
   E94 AT %M111.5 : Bool;
   E95 AT %M111.6 : Bool;
   E96 AT %M111.7 : Bool;
   E97 AT %M112.0 : Bool;   // Top carriage up (Top)
   E98 AT %M112.1 : Bool;   // Top carriage down (Top)
   E99 AT %M112.2 : Bool;   // Top carriage backward (Top)
   E100 AT %M112.3 : Bool;   // Top carriage forward (Top)
   E101 AT %M112.4 : Bool;   // Reading pallet height for top carriage (Top)
   E102 AT %M112.5 : Bool;   // Safety for top carriage movement (Top)
   E103 AT %M112.6 : Bool;   // Top film cutter forward (Top)
   E104 AT %M112.7 : Bool;   // Top film cutter backward (Top)
   E105 AT %M113.0 : Bool;   // Clamp to block top film closed (Top)
   E106 AT %M113.1 : Bool;   // Clamp to pull top film closed (Top)
   E107 AT %M113.2 : Bool;   // Top film ended sensor (Top)
   E108 AT %M113.3 : Bool;   // Safety for top carriage downward for infeed conveyor (Top)
   E109 AT %M113.4 : Bool;   // Safety for top carriage downward for outfeed conveyor (Top)
   E110 AT %M113.5 : Bool;   // Top carriage position under pressure plate (Top)
   E111 AT %M113.6 : Bool;   // Top carriage brake control (1 braked) (Top)
   E112 AT %M113.7 : Bool;
   E113 AT %M114.0 : Bool;
   E114 AT %M114.1 : Bool;
   E115 AT %M114.2 : Bool;
   E116 AT %M114.3 : Bool;
   E117 AT %M114.4 : Bool;   // SEGNALE PORTA TAGLIAFUOCO APERTA
   E118 AT %M114.5 : Bool;   // SEGNALE CHIUSURA PORTA TAGLIAFUOCO
   E119 AT %M114.6 : Bool;   // [B2782] CONTROLLO 1 POSIZIONAMENTO POS. 05
   E120 AT %M114.7 : Bool;   // [B2783] CONTROLLO 2 POSIZIONAMENTO POS. 05
   E121 AT %M115.0 : Bool;   // Pallet ready in infeed signal (Infeed signal)
   E122 AT %M115.1 : Bool;   // Ready to receive pallet from outfeed signal (Outfeed signal)
   E123 AT %M115.2 : Bool;   // End of pallet transfer signal (Outfeed signal)
   E124 AT %M115.3 : Bool;
   In_Pos1 AT %M116.0 : Bool;   // Conveyor pos.1 positioning support memory
   In_Forklift1 AT %M116.1 : Bool;   // Forklift presence conveyor pos.1 (support memory)
   In_Pos2 AT %M116.4 : Bool;   // Conveyor pos.2 positioning support memory
   In_Pos3 AT %M117.0 : Bool;   // Conveyor pos.3 positioning support memory
   A01 AT %M120.0 : Bool;   // Request to open door (Technoplat)
   A02 AT %M120.1 : Bool;   // Rele' on pilz chain (Technoplat)
   A03 AT %M120.2 : Bool;   // Emergency mode lamp (Technoplat)
   A04 AT %M120.3 : Bool;   // Automatic mode lamp (Technoplat)
   A05 AT %M120.4 : Bool;   // Film ended or broken lamp (Technoplat)
   A06 AT %M120.5 : Bool;   // Acoustic signal (Technoplat)
   A07 AT %M120.6 : Bool;   // Forward on table rotation inverter (Technoplat)
   A08_NotUsed AT %M120.7 : Bool;   // Speed selection (X2-S4I) on arm rotation inverter (Technoplat)
   A09_NotUsed AT %M121.0 : Bool;   // Speed selection (X3-S5I) on arm rotation inverter (Technoplat)
   A10 AT %M121.1 : Bool;   // Backward on table rotation inverter (Technoplat)
   A11 AT %M121.2 : Bool;   // Motor and brake for table rotation motor (Technoplat)
   A12 AT %M121.3 : Bool;   // Brake for table rotation motor (Technoplat)
   A13 AT %M121.4 : Bool;   // Forward on spool carriage(upward) and machine conveyor inverter (Technoplat)
   A14 AT %M121.5 : Bool;   // Backward on spool carriage(downward) and machine conveyor inverter (Technoplat)
   A15 AT %M121.6 : Bool;   // Spool carriage prestretch motor (Prestretch)
   A16 AT %M121.7 : Bool;   // Positioning command for OFF3 U201 (ON=normal functioning/OFF fast stop)
   A17_NotUsed AT %M122.0 : Bool;   // Pallet lifter upward(1)/downard (Lifter)
   A18_NotUsed AT %M122.1 : Bool;   // Pressure plate upward/downward(1) (Pressure plate)
   A19 AT %M122.2 : Bool;   // Opening/closing(1) single rope unit (Rope unit)
   A20 AT %M122.3 : Bool;   // Motor for spool carriage (Technoplat)
   A21_NotUsed AT %M122.4 : Bool;   // Jog1 speed for fast prestretch rool (Prestretch)
   A22_NotUsed AT %M122.5 : Bool;   // EN1 for fast prestretch rool (Prestretch)
   A23 AT %M122.6 : Bool;   // Opening/closing(1) lower (double) rope unit (Rope unit)
   A24 AT %M122.7 : Bool;   // Pressure plate upward (Technoplat pressure plate)
   A25 AT %M123.0 : Bool;   // Pressure plate downward (Technoplat pressure plate)
   A26 AT %M123.1 : Bool;   // Opening/closing(2) lower(double) rope unit (Rope unit)
   A27_NotUsed AT %M123.2 : Bool;
   A28 AT %M123.3 : Bool;   // LedBypass
   A29 AT %M123.4 : Bool;   // Enable (EN) for arm rotation and top inverter
   A30 AT %M123.5 : Bool;   // Motor for machine conveyor (Technoplat)
   A31_NotUsed AT %M123.6 : Bool;
   A32 AT %M123.7 : Bool;   // Ready to receive pallet from infeed signal reverse cycle
   A33 AT %M124.0 : Bool;   // End of pallet transfer from infeed signal reverse cycle
   A34 AT %M124.1 : Bool;   // Ready to receive pallet from infeed signal (Std signal)
   A35 AT %M124.2 : Bool;   // End of pallet transfer from infeed signal (Std signal)
   A36 AT %M124.3 : Bool;   // Pallet ready for outfeed signal (Std signal)
   A37_NotUsed AT %M124.4 : Bool;   // Motor for infeed conveyor (Conveyor)
   A38 AT %M124.5 : Bool;   // Machine in position signal (No conveyor signal)
   A39 AT %M124.6 : Bool;   // Wrapp ended signal (No conveyor signal)
   A40_NotUsed AT %M124.7 : Bool;
   A41_NotUsed AT %M125.0 : Bool;   // Film clamp upward (RingSpring clamp)
   A42_NotUsed AT %M125.1 : Bool;   // Film clamp downward (RingSpring clamp)
   A43_NotUsed AT %M125.2 : Bool;   // Film clamp opening(1)/closing (RingSpring clamp)
   A44 AT %M125.3 : Bool;   // Welder contrast upward(1)/downward (RingSpring clamp)
   A45_NotUsed AT %M125.4 : Bool;   // Welder unit upward(1)/downward (RingSpring clamp)
   A46 AT %M125.5 : Bool;   // Film cutter wire on (All clamp)
   A47 AT %M125.6 : Bool;   // Film welder on (All clamp)
   A48_NotUsed AT %M125.7 : Bool;   // Welder unit cooler (RingSpring clamp)
   A49 AT %M126.0 : Bool;   // Airblower for film tail (All clamp)
   A50 AT %M126.1 : Bool;   // Cutting and welding unit forward(1)/backward (Claw clamp)
   A51 AT %M126.2 : Bool;   // Film clamp opening (Claw clamp)
   A52 AT %M126.3 : Bool;   // Film clamp closing (Claw clamp)
   A53_NotUsed AT %M126.4 : Bool;   // Film clamp double closing (Claw clamp)
   A54_NotUsed AT %M126.5 : Bool;   // Welder unit forward(1)/backward (Claw clamp)
   A55_NotUsed AT %M126.6 : Bool;   // Film clamp carriage forward (Spring clamp)
   A56_NotUsed AT %M126.7 : Bool;   // Film clamp carriage backward (Spring clamp)
   A57 AT %M127.0 : Bool;   // Welder contrast forward (Contrast carriage)
   A58 AT %M127.1 : Bool;   // Welder contrast backward (Contrast carriage)
   A59 AT %M127.2 : Bool;   // Table position to open clamp during wrapping cycle
   A60 AT %M127.3 : Bool;
   A61 AT %M127.4 : Bool;
   A62 AT %M127.5 : Bool;
   A63 AT %M127.6 : Bool;   // Infeed safety barrier muting for muting by plc (Barrier)
   A64 AT %M127.7 : Bool;   // Outfeed safety barrier muting for muting by plc (Barrier)
   A65 AT %M128.0 : Bool;   // Signal ready to receive pallet from infeed (Infeed signal)
   A66 AT %M128.1 : Bool;   // Signal end of pallet transfer from infeed (Infeed signal)
   A67 AT %M128.2 : Bool;   // Signal pallet ready for outfeed (Outfeed signal)
   A68 AT %M128.3 : Bool;   // SEGNALE PRONTO PER CHIUSURA PORTA TAGLIAFUOCO
   A69 AT %M128.4 : Bool;
   A70 AT %M128.5 : Bool;
   A71 AT %M128.6 : Bool;
   A72 AT %M128.7 : Bool;
   A73 AT %M129.0 : Bool;
   A74 AT %M129.1 : Bool;
   A75 AT %M129.2 : Bool;   // Top carriage upward (Top)
   A76 AT %M129.3 : Bool;   // Top carriage downward (Top)
   A77 AT %M129.4 : Bool;   // Top carriage forward (Top)
   A78 AT %M129.5 : Bool;   // Top carriage backward (Top)
   A79 AT %M129.6 : Bool;   // Top cutter forward (Top)
   A80 AT %M129.7 : Bool;   // Top cutter backward (Top)
   A81 AT %M130.0 : Bool;   // Closing clamp to block top film (Top)
   A82 AT %M130.1 : Bool;   // Opening clamp to block top film (Top)
   A83 AT %M130.2 : Bool;   // Closing clamp to lift(pull) top film (Top)
   A84 AT %M130.3 : Bool;   // Opening clamp to lift(pull) top film (Top)
   A85 AT %M130.4 : Bool;   // Top carriage brake (Top)
   A86 AT %M130.5 : Bool;
   A87 AT %M130.6 : Bool;
   A88 AT %M130.7 : Bool;
   Clock01 AT %M255.0 : Bool;   // Clock 0,1 seconds (Period)
   Clock02 AT %M255.1 : Bool;   // Clock 0,2 seconds (Period)
   Clock04 AT %M255.2 : Bool;   // Clock 0,4 seconds (Period)
   Clock05 AT %M255.3 : Bool;   // Clock 0,5 seconds (Period)
   Clock08 AT %M255.4 : Bool;   // Clock 0,8 seconds (Period)
   Clock10 AT %M255.5 : Bool;   // Clock 1,0 seconds (Period)
   Clock16 AT %M255.6 : Bool;   // Clock 1,6 seconds (Period)
   Clock20 AT %M255.7 : Bool;   // Clock 2,0 seconds (Period)
   MB0 AT %MB0 : Byte;   // Machine cycle (1) byte
   MB1 AT %MB1 : Byte;   // Machine cycle (2) byte
   MW2 AT %MW2 : Word;   // Machine cycle (3) word
   MB5 AT %MB5 : Byte;   // Top cycle (1) byte
   MW6 AT %MW6 : Word;   // Top cycle (2) word
   MW8 AT %MW8 : Word;   // Top film ended cycle word
   Tag_9 AT %M8.7 : Bool;
   MB16 AT %MB16 : Byte;   // Conveyor cycle byte
   MB17 AT %MB17 : Byte;   // Pallet load cycle byte
   MB20 AT %MB20 : Byte;   // Claw clamp HS40 cycle byte
   MB24 AT %MB24 : Byte;
   MB30 AT %MB30 : Byte;   // Film broken cycle byte
   MB32 AT %MB32 : Byte;   // Film broken cycle 1 byte
   In_Forklift2 AT %M116.5 : Bool;   // Forklift presence conveyor pos.2 (support memory)
   V50_0 AT %M50.0 : Bool;   // Support for end of transfer signal
   V50_2 AT %M50.2 : Bool;   // Transit memory pos1->pos2
   V51_2 AT %M51.2 : Bool;   // Memory to exclude wrapping in pos 2
   In_Pos4 AT %M117.4 : Bool;   // Conveyor pos.4 positioning support memory
   In_Forklift4 AT %M117.5 : Bool;   // Forklift presence conveyor pos.4 (support memory)
   V52_0 AT %M52.0 : Bool;   // Transit memory pos3->pos4
   V50_4 AT %M50.4 : Bool;   // Transit memory pos3->pos4
   V52_1 AT %M52.1 : Bool;   // Outfeed conveyor pos.4 unload
   V50_5 AT %M50.5 : Bool;   // Transit memory pos4->pos5
   "M1.4_N" AT %M200.0 : Bool;   // Negative edge M1.4
   V50_3 AT %M50.3 : Bool;   // Transit memory pos2->pos3
   In_Forklift3 AT %M117.1 : Bool;   // Forklift presence conveyor pos.3 (support memory)
   Off AT %M12.6 : Bool;   // Bit always off
   U201_Start AT %M161.0 : Bool;
   U201_Ack AT %M161.1 : Bool;
   U201_Rev AT %M161.2 : Bool;
   U221_Start AT %M161.3 : Bool;
   U221_Ack AT %M161.4 : Bool;
   U221_Rev AT %M161.5 : Bool;
   U241_Start AT %M161.6 : Bool;
   U241_Ack AT %M161.7 : Bool;
   U241_Rev AT %M162.0 : Bool;
   U261_Start AT %M162.1 : Bool;
   U261_Ack AT %M162.2 : Bool;
   U261_Rev AT %M162.3 : Bool;
   U321_Start AT %M162.4 : Bool;
   U321_Ack AT %M162.5 : Bool;
   U321_Rev AT %M162.6 : Bool;
   U201_OFF1 AT %M170.0 : Bool;
   U201_OFF3 AT %M170.1 : Bool;
   U321_OFF1 AT %M170.2 : Bool;
   U321_OFF3 AT %M170.3 : Bool;
   InverterFail AT %M163.0 : Bool;   // Inverter Fault/Alarm - Anomalia/Avviso
   InverterFault AT %M163.1 : Bool;   // Inverter Fault (F) - Anomalia
   InverterAlarm AT %M163.2 : Bool;   // Inverter Alarm (A) - Avviso
   PrestNewValue AT %M160.0 : Bool;
   System_Byte AT %MB254 : Byte;
   FirstScan AT %M254.0 : Bool;
   DiagStatusUpdate AT %M254.1 : Bool;
   AlwaysTRUE AT %M254.2 : Bool;
   AlwaysFALSE AT %M254.3 : Bool;
   U201_Start_ARM AT %M170.6 : Bool;
   U201_Start_RUL AT %M170.7 : Bool;
   U201_Feedback AT %M171.0 : Bool;   // Feedback motori sotto inverter U201 (braccio/rull.CM)
   U221_Feedback AT %M171.1 : Bool;   // Feedback motore sotto inverter U221 (carrello)
   U241_Feedback AT %M171.2 : Bool;   // Feedback motore sotto inverter U241 (tiro)
   U261_Feedback AT %M171.3 : Bool;   // Feedback motore sotto inverter U261 (prestiro)
   Tag_14 AT %M13.2 : Bool;
   Tag_10 AT %M14.5 : Bool;
   CELLA AT %MW145 : Int;   // Valore cella di carico (modbus)
   ResetLoadCell AT %M144.7 : Bool;   // "DB100_Display".ResetLoadCell
   ERR AT %MD155 : DInt;   // Errore (SP-feedback)
   PROVA AT %MD150 : DWord;
   BitClock1 AT %M143.1 : Bool;   // Impulso ogni 20ms (OB30)
   BitClock2 AT %M143.2 : Bool;   // Impulso ogni 100ms (OB30 x5)
   In_Pos5 AT %M117.6 : Bool;   // Conveyor pos.5 positioning support memory
   In_Pos6 AT %M117.7 : Bool;   // Conveyor pos.6 positioning support memory
   In_Pos7 AT %M118.0 : Bool;   // Conveyor pos.7 positioning support memory
   In_Pos8 AT %M118.1 : Bool;   // Conveyor pos.8 positioning support memory
   V50_7 AT %M50.7 : Bool;   // Transit memory pos7->pos8
   V51_0 AT %M51.0 : Bool;   // Outfeed conveyor pos.8 unload
   V51_3 AT %M51.3 : Bool;   // Memory to exclude wrapping in pos 3
   V51_4 AT %M51.4 : Bool;   // Memory to exclude wrapping in pos 4
   V51_5 AT %M51.5 : Bool;   // Memory to exclude wrapping in pos 5
   Centrador_Aberto_1 AT %I8.0 : Bool;
   Centrador_Aberto_2 AT %I8.1 : Bool;
   Palete_Centrada_1 AT %I8.2 : Bool;
   Palete_Centrada_2 AT %I8.3 : Bool;
   Tag_1 AT %Q8.3 : Bool;
   "M13.0" AT %M13.0 : Bool;
END_VAR

TYPE "APP"
// stored: IsFailsafeCompliant false
   STRUCT
      PID_ComponenteProporzionale : DInt;
      PID_ComponenteIntegrale : DInt;
      PID_ComponenteDerivativa : DInt;
      Tiro : Int;   // Valore di tiro richiesto: 1-100 => 1-100% Setup 1, 101-200 => 1-100% Setup 2, 0 => Azzera regolatore
      Tiro1 : Int;
      Tiro2 : Int;
      TiroPrecedente : Int;   // Valore di tiro richiesto istante (n-1)
      TiroAppoggio : Int;
      ErroreAttuale : Int;   // Errore istante (n)
      ErrorePrecedente : Int;   // Errore istante (n-1)
      PID_Kp : Int;   // Kp in uso nel PID
      PID_Ki : Int;   // Ki in uso nel PID
      PID_Kd : Int;   // Kd in uso nel PID
      SetpointTiro : Int;   // Valore di setpoint del PID
      SetpointTiroRampa : Int;   // Valore di setpoint del PID iniziale a rampa
      TransitorioInizialeFase1 : Int;   // Indica che si deve eseguire la rampa iniziale (Fase 1)
      TransitorioFase3 : Int;   // Indica che si deve eseguire la rampa da velocita' alta a media (Fase 3)
      TransitorioFase4 : Int;   // Indica che si deve eseguire la rampa da velocita' media a bassa (Fase 4)
      VelocitaRotazione : Int;   // Velocita' di rotazione richiesta
      VelocitaRotazioneFase2 : Int;   // Velocita' di rotazione richiesta durante la Fase 2
      VelocitaRotazioneAppoggio1 : Int;
      VelocitaRotazioneAppoggio2 : Int;
      Fase1OneShoot : Int;   // Indica che sono appena entrato nella fase di traansitorio di accelerazione (Fase 1)
      Fase2OneShoot : Int;   // Indica che sono appena entrato nella fase di transitorio iniziale (Fase 2)
      Fase3OneShoot : Int;   // Indica che sono appena entrato nella fase di transitorio di velocita' alta - media (Fase 3)
      Fase4OneShoot : Int;   // Indica che sono appena entrato nella fase di transitorio di velocita' media - bassa (Fase 4)
      ArrestoRepentinoOneShoot : Int;   // Indica che sono appena entrato nella fase di arresto repentino
      TiroFase1 : Int;   // Indica il tiro nella Fase 1 usato nella Fase 2
      TempIntero : Int;
      Fase : Int;
      BallerinoPrecedente : Array[0..2] of Int;   // Valore del ballerino negli istanti precedenti
      LimiteComponenteIntegrale : Int;   // Limite della componente integrale durante la transizione dalla velocita alta a media (Fase 3) e dalla media a bassa (Fase 4)
      TiroRichiesto : Int;   // Valore di tiro compreso fra 1 e 100 richiesto dalla logica di controllo
      TimerArrestoRepentino : Int;   // Timer per arresto repentino.
      TiroMinimoArrestoRepentino : Int;   // Tiro minimo durante un'arresto repentino
      VariazioneTiro : Int;   // Variazione del tiro film (ballerino)
      TimerFase2 : Int;   // Timer usato nella Fase 2 per arrestare i rulli in caso di rottura film
      TempoRotturaFilm : Int;   // Tempo rottura film in numero di scansioni (1 scansione ogni 30msec)
      TimerFase4 : Int;   // Timer per Fase 4
      TiroMinimoFase4 : Int;   // Tiro minimo durante la Fase 4 di arresto
      PID_Uscita : DInt;   // Valore di uscita del PID
      PrestiroRichiesto : DInt;   // Valore di prestiro richiesto. Valore compreso fra 0 e 500
      PrestiroAppoggio : Real;
   END_STRUCT;
END_TYPE

TYPE "DatiProgramma"
// stored: IsFailsafeCompliant false
   STRUCT
      Wrapping : Bool;   // Wrapping (0=Excluded 1=Included)
      TopLenght : Int;   // Top film lenght
      TopRelease : Int;   // Top carriage release position
      TopDown : Int;   // Top carriage downward to release top film
      Top : Int;   // Top cycle (1=Excluded 2=Before 3=Waterp-2 4=Waterp-3 5=Waterp-4)
      PressurePTime : Int;   // Time for pressure plate downward
      LifterTime : Int;   // Time for pallet lifter upward
      RevOverContrast : Int;   // Revolution over welder contrast
      RopeEndCycle : Byte;   // Rope type at end of cycle (Program)
      Spare4 : Byte;
      RopeTime : Int;   // Delay for rope unit opened
      RevOverClamp : Int;   // Revolution over clamp
      FilmForceFinalRev : Int;   // Film force on the final revolutions
      FilmPrestretchFinalRev : Int;   // Film prestretch on the final revolutions
      ArmSpeed : Int;   // Arm rotation speed (%*10)
      CarriageDown4Top : Int;   // Spool carriage downward for top cycle
      TopDownTime : Int;   // Top carriage downward for top cycle
      LapsUnderTop : Int;   // Revolutions under top film
      Spare6 : Int;   // Spare
      Spare7 : Int;   // Spare
      Spare8 : Int;   // Spare
      Spare9 : Int;   // Spare
      Spare10 : Int;   // Spare
      Spare11 : Int;   // Spare
      Spare12 : Int;   // Spare
      Overlap0_1 : Int := 0;   // Film overlap spool carriage height 0->1
      Height1 : Int := 0;   // Spool carriage height 1 (mm)
      Landmark1 : Bool := false;   // Landmark for spool carriage height 1 (0=Bottom 1=Top)
      Lifter1 : Bool := false;   // Pallet lifter for spool carriage height 1
      SpareBit1H1 : Bool := false;   // Spare bit for spool carriage height 1 (Program)
      Airblower1 : Bool := false;   // Airblower on film tail for spool carriage height 1 (0=Excluded 1=Included)
      NextStep1 : Bool := false;   // Next step for spool carriage height 1 (0=End 1=Next)
      PressureP1 : Bool := false;   // Pressure plate for spool carriage height 1 (0=Excluded 1=Included)
      SpareByte2H1 : Byte := 16#0;   // Spare byte for spool carriage height 1
      Revolution1 : Int := 0;   // Revolutions for spool carriage height 1
      RopeUnit1_1 : Byte := 16#0;   // Rope unit for spool carriage height 1 (1=Excluded 2=Inc 3=Inc during)
      RopeUnit1_2 : Byte := 16#0;   // Rope unit for spool carriage height 1 (1=Excluded 2=Inc 3=Inc during)
      FilmForce1 : Int := 0;   // Film force for spool carriage height 1
      FilmPrestretch1 : Int := 0;   // Film prestretch for spool carriage height 1
      Spare3H1 : Int := 0;   // Spare for spool carriage height 1
      Spare49 : Int := 0;   // Spare
      Spare50 : Int := 0;   // Spare
      Spare51 : Int := 0;   // Spare
      Spare52 : Int := 0;   // Spare
      Spare53 : Int := 0;   // Spare
      Overlap1_2 : Int := 0;   // Film overlap spool carriage height 1->2
      Height2 : Int := 0;   // Spool carriage height 2 (mm)
      Landmark2 : Bool := false;   // Landmark for spool carriage height 2 (0=Bottom 1=Top)
      Lifter2 : Bool := false;   // Pallet lifter for spool carriage height 2
      SpareBit1H2 : Bool := false;   // Spare bit for spool carriage height 2
      Airblower2 : Bool := false;   // Airblower on film tail for spool carriage height 2 (0=Excluded 1=Included)
      NextStep2 : Bool := false;   // Next step for spool carriage height 2 (0=End 1=Next)
      PressureP2 : Bool := false;   // Pressure plate for spool carriage height 2 (0=Excluded 1=Included)
      SpareByte2H2 : Byte := 16#0;   // Spare byte for spool carriage height 2
      Revolution2 : Int := 0;   // Revolutions for spool carriage height 2
      RopeUnit2_1 : Byte := 16#0;   // Rope unit for spool carriage height 2 (1=Excluded 2=Inc 3=Inc during)
      RopeUnit2_2 : Byte := 16#0;   // Rope unit for spool carriage height 2 (1=Excluded 2=Inc 3=Inc during)
      FilmForce2 : Int := 0;   // Film force for spool carriage height 2
      FilmPrestretch2 : Int := 0;   // Film prestretch for spool carriage height 2
      Spare3H2 : Int := 0;   // Spare for spool carriage height 2
      Spare54 : Int := 0;   // Spare
      Spare55 : Int := 0;   // Spare
      Spare56 : Int := 0;   // Spare
      Spare57 : Int := 0;   // Spare
      Spare58 : Int := 0;   // Spare
      Overlap2_3 : Int := 0;   // Film overlap spool carriage height 2->3
      Height3 : Int := 0;   // Spool carriage height 3 (mm)
      Landmark3 : Bool := false;   // Landmark for spool carriage height 3 (0=Bottom 1=Top)
      Lifter3 : Bool := false;   // Pallet lifter for spool carriage height 3
      SpareBit1H3 : Bool := false;   // Spare bit for spool carriage height 3
      Airblower3 : Bool := false;   // Airblower on film tail for spool carriage height 3 (0=Excluded 1=Included)
      NextStep3 : Bool := false;   // Next step for spool carriage height 3 (0=End 1=Next)
      PressureP3 : Bool := false;   // Pressure plate for spool carriage height 3 (0=Excluded 1=Included)
      SpareByte2H3 : Byte := 16#0;   // Spare byte for spool carriage height 3
      Revolution3 : Int := 0;   // Revolutions for spool carriage height 3
      RopeUnit3_1 : Byte := 16#0;   // Rope unit for spool carriage height 3 (1=Excluded 2=Inc 3=Inc during)
      RopeUnit3_2 : Byte := 16#0;   // Rope unit for spool carriage height 3 (1=Excluded 2=Inc 3=Inc during)
      FilmForce3 : Int := 0;   // Film force for spool carriage height 3
      FilmPrestretch3 : Int := 0;   // Film prestretch for spool carriage height 3
      Spare3H3 : Int := 0;   // Spare for spool carriage height 3
      Spare59 : Int := 0;   // Spare
      Spare60 : Int := 0;   // Spare
      Spare61 : Int := 0;   // Spare
      Spare62 : Int := 0;   // Spare
      Spare63 : Int := 0;   // Spare
      Overlap3_4 : Int := 0;   // Film overlap spool carriage height 3->4
      Height4 : Int := 0;   // Spool carriage height 4 (mm)
      Landmark4 : Bool := false;   // Landmark for spool carriage height 4 (0=Bottom 1=Top)
      Lifter4 : Bool := false;   // Pallet lifter for spool carriage height 4
      SpareBit1H4 : Bool := false;   // Spare bit for spool carriage height 4
      Airblower4 : Bool := false;   // Airblower on film tail for spool carriage height 4 (0=Excluded 1=Included)
      NextStep4 : Bool := false;   // Next step for spool carriage height 4 (0=End 1=Next)
      PressureP4 : Bool := false;   // Pressure plate for spool carriage height 4 (0=Excluded 1=Included)
      SpareByte2H4 : Byte := 16#0;   // Spare byte for spool carriage height 4
      Revolution4 : Int := 0;   // Revolutions for spool carriage height 4
      RopeUnit4_1 : Byte := 16#0;   // Rope unit for spool carriage height 4 (1=Excluded 2=Inc 3=Inc during)
      RopeUnit4_2 : Byte := 16#0;   // Rope unit for spool carriage height 4 (1=Excluded 2=Inc 3=Inc during)
      FilmForce4 : Int := 0;   // Film force for spool carriage height 4
      FilmPrestretch4 : Int := 0;   // Film prestretch for spool carriage height 4
      Spare3H4 : Int := 0;   // Spare for spool carriage height 4
      Spare64 : Int := 0;   // Spare
      Spare65 : Int := 0;   // Spare
      Spare66 : Int := 0;   // Spare
      Spare67 : Int := 0;   // Spare
      Spare68 : Int := 0;   // Spare
      Overlap4_5 : Int := 0;   // Film overlap spool carriage height 4->5
      Height5 : Int := 0;   // Spool carriage height 5 (mm)
      Landmark5 : Bool := false;   // Landmark for spool carriage height 5 (0=Bottom 1=Top)
      Lifter5 : Bool := false;   // Pallet lifter for spool carriage height 5
      SpareBit1H5 : Bool := false;   // Spare bit for spool carriage height 5
      Airblower5 : Bool := false;   // Airblower on film tail for spool carriage height 5 (0=Excluded 1=Included)
      NextStep5 : Bool := false;   // Next step for spool carriage height 5 (0=End 1=Next)
      PressureP5 : Bool := false;   // Pressure plate for spool carriage height 5 (0=Excluded 1=Included)
      SpareByte2H5 : Byte := 16#0;   // Spare byte for spool carriage height 5
      Revolution5 : Int := 0;   // Revolutions for spool carriage height 5
      RopeUnit5_1 : Byte := 16#0;   // Rope unit for spool carriage height 5 (1=Excluded 2=Inc 3=Inc during)
      RopeUnit5_2 : Byte := 16#0;   // Rope unit for spool carriage height 5 (1=Excluded 2=Inc 3=Inc during)
      FilmForce5 : Int := 0;   // Film force for spool carriage height 5
      FilmPrestretch5 : Int := 0;   // Film prestretch for spool carriage height 5
      Spare3H5 : Int := 0;   // Spare for spool carriage height 5
      Spare69 : Int := 0;   // Spare
      Spare70 : Int := 0;   // Spare
      Spare71 : Int := 0;   // Spare
      Spare72 : Int := 0;   // Spare
      Spare73 : Int := 0;   // Spare
      Overlap5_6 : Int := 0;   // Film overlap spool carriage height 5->6
      Height6 : Int := 0;   // Spool carriage height 6 (mm)
      Landmark6 : Bool := false;   // Landmark for spool carriage height 6 (0=Bottom 1=Top)
      Lifter6 : Bool := false;   // Pallet lifter for spool carriage height 6
      SpareBit1H6 : Bool := false;   // Spare bit for spool carriage height 6
      Airblower6 : Bool := false;   // Airblower on film tail for spool carriage height 6 (0=Excluded 1=Included)
      NextStep6 : Bool := false;   // Next step for spool carriage height 6 (0=End 1=Next)
      PressureP6 : Bool := false;   // Pressure plate for spool carriage height 6 (0=Excluded 1=Included)
      SpareByte2H6 : Byte := 16#0;   // Spare byte for spool carriage height 6
      Revolution6 : Int := 0;   // Revolutions for spool carriage height 6
      RopeUnit6_1 : Byte := 16#0;   // Rope unit for spool carriage height 6 (1=Excluded 2=Inc 3=Inc during)
      RopeUnit6_2 : Byte := 16#0;   // Rope unit for spool carriage height 6 (1=Excluded 2=Inc 3=Inc during)
      FilmForce6 : Int := 0;   // Film force for spool carriage height 6
      FilmPrestretch6 : Int := 0;   // Film prestretch for spool carriage height 6
      Spare3H6 : Int := 0;   // Spare for spool carriage height 6
      Spare74 : Int := 0;   // Spare
      Spare75 : Int := 0;   // Spare
      Spare76 : Int := 0;   // Spare
      Spare77 : Int := 0;   // Spare
      Spare78 : Int := 0;   // Spare
      Overlap6_7 : Int := 0;   // Film overlap spool carriage height 6->7
      Height7 : Int := 0;   // Spool carriage height 7 (mm)
      Landmark7 : Bool := false;   // Landmark for spool carriage height 7 (0=Bottom 1=Top)
      Lifter7 : Bool := false;   // Pallet lifter for spool carriage height 7
      SpareBit1H7 : Bool := false;   // Spare bit for spool carriage height 7
      Airblower7 : Bool := false;   // Airblower on film tail for spool carriage height 7 (0=Excluded 1=Included)
      NextStep7 : Bool := false;   // Next step for spool carriage height 7 (0=End 1=Next)
      PressureP7 : Bool := false;   // Pressure plate for spool carriage height 7 (0=Excluded 1=Included)
      SpareByte2H7 : Byte := 16#0;   // Spare byte for spool carriage height 7
      Revolution7 : Int := 0;   // Revolutions for spool carriage height 7
      RopeUnit7_1 : Byte := 16#0;   // Rope unit for spool carriage height 7 (1=Excluded 2=Inc 3=Inc during)
      RopeUnit7_2 : Byte := 16#0;   // Rope unit for spool carriage height 7 (1=Excluded 2=Inc 3=Inc during)
      FilmForce7 : Int := 0;   // Film force for spool carriage height 7
      FilmPrestretch7 : Int := 0;   // Film prestretch for spool carriage height 7
      Spare3H7 : Int := 0;   // Spare for spool carriage height 7
      Spare79 : Int := 0;   // Spare
      Spare80 : Int := 0;   // Spare
      Spare81 : Int := 0;   // Spare
      Spare82 : Int := 0;   // Spare
      Spare83 : Int := 0;   // Spare
      Overlap7_8 : Int := 0;   // Film overlap spool carriage height 7->8
      Height8 : Int := 0;   // Spool carriage height 8 (mm)
      Landmark8 : Bool := false;   // Landmark for spool carriage height 8 (0=Bottom 1=Top)
      Lifter8 : Bool := false;   // Pallet lifter for spool carriage height 8
      SpareBit1H8 : Bool := false;   // Spare bit for spool carriage height 8
      Airblower8 : Bool := false;   // Airblower on film tail for spool carriage height 8 (0=Excluded 1=Included)
      NextStep8 : Bool := false;   // Next step for spool carriage height 8 (0=End 1=Next)
      PressureP8 : Bool := false;   // Pressure plate for spool carriage height 8 (0=Excluded 1=Included)
      SpareByte2H8 : Byte := 16#0;   // Spare byte for spool carriage height 8
      Revolution8 : Int := 0;   // Revolutions for spool carriage height 8
      RopeUnit8_1 : Byte := 16#0;   // Rope unit for spool carriage height 8 (1=Excluded 2=Inc 3=Inc during)
      RopeUnit8_2 : Byte := 16#0;   // Rope unit for spool carriage height 8 (1=Excluded 2=Inc 3=Inc during)
      FilmForce8 : Int := 0;   // Film force for spool carriage height 8
      FilmPrestretch8 : Int := 0;   // Film prestretch for spool carriage height 8
      Spare3H8 : Int := 0;   // Spare for spool carriage height 8
      Spare84 : Int := 0;   // Spare
      Spare85 : Int := 0;   // Spare
      Spare86 : Int := 0;   // Spare
      Spare87 : Int := 0;   // Spare
      Spare88 : Int := 0;   // Spare
      Overlap8_9 : Int := 0;   // Film overlap spool carriage height 8->9
      Height9 : Int := 0;   // Spool carriage height 9 (mm)
      Landmark9 : Bool := false;   // Landmark for spool carriage height 9 (0=Bottom 1=Top)
      Lifter9 : Bool := false;   // Pallet lifter for spool carriage height 9
      SpareBit1H9 : Bool := false;   // Spare bit for spool carriage height 9
      Airblower9 : Bool := false;   // Airblower on film tail for spool carriage height 9 (0=Excluded 1=Included)
      NextStep9 : Bool := false;   // Next step for spool carriage height 9 (0=End 1=Next)
      PressureP9 : Bool := false;   // Pressure plate for spool carriage height 9 (0=Excluded 1=Included)
      SpareByte2H9 : Byte := 16#0;   // Spare byte for spool carriage height 9
      Revolution9 : Int := 0;   // Revolutions for spool carriage height 9
      RopeUnit9_1 : Byte := 16#0;   // Rope unit for spool carriage height 9 (1=Excluded 2=Inc 3=Inc during)
      RopeUnit9_2 : Byte := 16#0;   // Rope unit for spool carriage height 9 (1=Excluded 2=Inc 3=Inc during)
      FilmForce9 : Int := 0;   // Film force for spool carriage height 9
      FilmPrestretch9 : Int := 0;   // Film prestretch for spool carriage height 9
      Spare3H9 : Int := 0;   // Spare for spool carriage height 9
      Spare89 : Int := 0;   // Spare
      Spare90 : Int := 0;   // Spare
      Spare91 : Int := 0;   // Spare
      Spare92 : Int := 0;   // Spare
      Spare93 : Int := 0;   // Spare
      Overlap9_10 : Int := 0;   // Film overlap spool carriage height 9->10
      Height10 : Int := 0;   // Spool carriage height 10 (mm)
      Landmark10 : Bool := false;   // Landmark for spool carriage height 10 (0=Bottom 1=Top)
      Lifter10 : Bool := false;   // Pallet lifter for spool carriage height 10
      SpareBit1H10 : Bool := false;   // Spare bit for spool carriage height 10
      Airblower10 : Bool := false;   // Airblower on film tail for spool carriage height 10 (0=Excluded 1=Included)
      NextStep10 : Bool := false;   // Next step for spool carriage height 10 (0=End 1=Next)
      PressureP10 : Bool := false;   // Pressure plate for spool carriage height 10 (0=Excluded 1=Included)
      SpareByte2H10 : Byte := 16#0;   // Spare byte for spool carriage height 10
      Revolution10 : Int := 0;   // Revolutions for spool carriage height 10
      RopeUnit10_1 : Byte := 16#0;   // Rope unit for spool carriage height 10 (1=Excluded 2=Inc 3=Inc during)
      RopeUnit10_2 : Byte := 16#0;   // Rope unit for spool carriage height 10 (1=Excluded 2=Inc 3=Inc during)
      FilmForce10 : Int := 0;   // Film force for spool carriage height 10
      FilmPrestretch10 : Int := 0;   // Film prestretch for spool carriage height 10
      Spare3H10 : Int := 0;   // Spare for spool carriage height 10
      Spare94 : Int := 0;   // Spare
      Spare95 : Int := 0;   // Spare
      Spare96 : Int := 0;   // Spare
      Spare97 : Int := 0;   // Spare
      Spare98 : Int := 0;   // Spare
      Overlap10_11 : Int := 0;   // Film overlap spool carriage height 10->11
      Height11 : Int := 0;   // Spool carriage height 11 (mm)
      Landmark11 : Bool := false;   // Landmark for spool carriage height 11 (0=Bottom 1=Top)
      Lifter11 : Bool := false;   // Pallet lifter for spool carriage height 11
      SpareBit1H11 : Bool := false;   // Spare bit for spool carriage height 11
      Airblower11 : Bool := false;   // Airblower on film tail for spool carriage height 11 (0=Excluded 1=Included)
      NextStep11 : Bool := false;   // Next step for spool carriage height 11 (0=End 1=Next)
      PressureP11 : Bool := false;   // Pressure plate for spool carriage height 11 (0=Excluded 1=Included)
      SpareByte2H11 : Byte := 16#0;   // Spare byte for spool carriage height 11
      Revolution11 : Int := 0;   // Revolutions for spool carriage height 11
      RopeUnit11_1 : Byte := 16#0;   // Rope unit for spool carriage height 11 (1=Excluded 2=Inc 3=Inc during)
      RopeUnit11_2 : Byte := 16#0;   // Rope unit for spool carriage height 11 (1=Excluded 2=Inc 3=Inc during)
      FilmForce11 : Int := 0;   // Film force for spool carriage height 11
      FilmPrestretch11 : Int := 0;   // Film prestretch for spool carriage height 11
      Spare3H11 : Int := 0;   // Spare for spool carriage height 11
      Spare99 : Int := 0;   // Spare
      Spare100 : Int := 0;   // Spare
      Spare101 : Int := 0;   // Spare
      Spare102 : Int := 0;   // Spare
      Spare103 : Int := 0;   // Spare
      Overlap11_12 : Int := 0;   // Film overlap spool carriage height 11->12
      Height12 : Int := 0;   // Spool carriage height 12 (mm)
      Landmark12 : Bool := false;   // Landmark for spool carriage height 12 (0=Bottom 1=Top)
      Lifter12 : Bool := false;   // Pallet lifter for spool carriage height 12
      SpareBit1H12 : Bool := false;   // Spare bit for spool carriage height 12
      Airblower12 : Bool := false;   // Airblower on film tail for spool carriage height 12 (0=Excluded 1=Included)
      NextStep12 : Bool := false;   // Next step for spool carriage height 12 (0=End 1=Next)
      PressureP12 : Bool := false;   // Pressure plate for spool carriage height 12 (0=Excluded 1=Included)
      SpareByte2H12 : Byte := 16#0;   // Spare byte for spool carriage height 12
      Revolution12 : Int := 0;   // Revolutions for spool carriage height 12
      RopeUnit12_1 : Byte := 16#0;   // Rope unit for spool carriage height 12 (1=Excluded 2=Inc 3=Inc during)
      RopeUnit12_2 : Byte := 16#0;   // Rope unit for spool carriage height 12 (1=Excluded 2=Inc 3=Inc during)
      FilmForce12 : Int := 0;   // Film force for spool carriage height 12
      FilmPrestretch12 : Int := 0;   // Film prestretch for spool carriage height 12
      Spare3H12 : Int := 0;   // Spare for spool carriage height 12
      Spare104 : Int := 0;   // Spare
      Spare105 : Int := 0;   // Spare
      Spare106 : Int := 0;   // Spare
      Spare107 : Int := 0;   // Spare
      Spare108 : Int := 0;   // Spare
   END_STRUCT;
END_TYPE

TYPE "InverterData"
// stored: IsFailsafeCompliant false
   STRUCT
      control_word : Word;
      setpoint : Real;
      ref_quantity : Struct
         speed_p2000 : Real;
         current_p2002 : Real;
         torque_p2003 : Real;
      END_STRUCT;
      status_word : Word;
      actual_speed : Real;
      actual_current : Real;
      actual_torque : Real;
      actual_alarm : Word;
      actual_fault : Word;
      RETVAL_RD : Word;
      RETVAL_WR : Word;
   END_STRUCT;
END_TYPE

TYPE "M20"
// stored: IsFailsafeCompliant false
   STRUCT
      M20_P00 : Int;   // Tipo di prestiro
      M20_P01 : Int;   // Coefficiente proporzionale per il regolatore PID
      M20_P02 : Int;   // Coefficiente integrale (Fase1 e Fase2) per il regolatore PID
      M20_P03 : Int;   // Coefficiente derivativo per il regolatore PID
      M20_P04 : Int;   // Coefficiente integrale (Fase3 e Fase4) per il regolatore PID
      M20_P05 : Int;   // Rampa di accelerazione per il tiro durante la Fase1
      M20_P06 : Int;   // Limite componente integrale nel transitorio dalla Fase2 alla Fase3
      M20_P07 : Int;   // Limite componente integrale nel transitorio dalla Fase3 alla Fase4
      M20_P08 : Int;   // Valore minimo ingresso analogico
      M20_P09 : Int;   // Valore massimo ingresso analogico
      M20_P10 : Int;   // Prestiro naturale dovuto al rapporto di riduzione
      M20_P11 : Int;   // Velocità per il jog in manuale dei rulli di prestiro
      M20_P12 : Int;   // Offset del rullo lento 10 equivale a 0
      M20_P13 : Int;   // Jog di velocità durante la partenza del braccio
      M20_P14 : Int;   // Tiro minimo durante la Fase4 di arresto e durante un arresto repentino
      M20_P15 : Int;   // Tempo (in decimi di secondo) dopo il quale i rulli si fermano per rottura film
      M20_P20 : Int;   // Velocità indicata da plc per la rotazione braccio e il carrello top
      M20_P21 : Int;   // Velocità indicata da plc per il carrello di prestiro e il trasporto di centro macchina
      M20_P22 : Int;   // Tiro indicato da plc
      M20_P23 : Int;   // Prestiro indicato da plc
      M20_P24 : Int;   // Valore di ingresso analogico AI0
      M20_P25 : Int;   // Tiro richiesto da plc compreso fra 0 e 100
   END_STRUCT;
END_TYPE

TYPE "PID"
// stored: IsFailsafeCompliant false
   STRUCT
      proporzionale : DInt;
      integrativo : DInt;
      segnale : DInt;
      maxSegnale : Int;
      minSegnale : Int;
      setPointShow : UInt;
      tiro : UInt;
      vParP : UInt;
      vParI : UInt;
      svuota : Bool;
      attiva : Bool;
      setTiro : Bool;
      "timer" : Time;
   END_STRUCT;
END_TYPE

TYPE "ProgramDataGreyBar"
// stored: IsFailsafeCompliant false
   STRUCT
      Overlap : Int;   // Film overlap
      Height : Int;   // Spool carriage height (mm)
      Landmark : Bool;   // Landmark (0=Bottom 1=Top)
      Lifter : Bool;   // Pallet lifter
      SpareBit1 : Bool;   // Spare
      Airblower : Bool;   // Airblower on film tail (0=Excluded 1=Included)
      NextStep : Bool;   // Next step (0=End 1=Next)
      PressureP : Bool;   // Pressure plate (0=Excluded 1=Included)
      SpareByte1 : Byte;   // Spare
      Revolution : Int;   // Revolutions
      RopeUnitUpper : Byte;   // Upper rope unit (1=Exc 2=Inc 3=Inc during)
      RopeUnitLower : Byte;   // Lower rope unit (1=Exc 2=Inc 3=Inc during)
      FilmForce : Int;   // Film force
      FilmPrestretch : Int;   // Film prestretch
      SpareWord1 : Int;   // Spare
      SpareWord2 : Int;   // Spare
      SpareWord3 : Int;   // Spare
      SpareWord4 : Int;   // Spare
      SpareWord5 : Int;   // Spare
      SpareWord6 : Int;   // Spare
   END_STRUCT;
END_TYPE

DATA_BLOCK "DB01_Osr"   // DB1
{ S7_Optimized_Access := 'FALSE' }
AUTHOR : Robopac
VERSION : 0.0
// stored: AutoNumber false, IsOnlyStoredInLoadMemory false, IsWriteProtectedInAS false
   VAR RETAIN
      osr1 : Bool := TRUE;   // Used
      osr2 : Bool := FALSE;   // Used
      osr3 : Bool := FALSE;   // Used
      osr4 : Bool := FALSE;   // Used
      osr5 : Bool := FALSE;   // Used
      osr6 : Bool := TRUE;   // Used
      osr7 : Bool := TRUE;   // Used
      osr8 : Bool := FALSE;   // Used
      osr9 : Bool := TRUE;   // Used
      osr10 : Bool := FALSE;   // Used
      osr11 : Bool := FALSE;   // Used
      osr12 : Bool := FALSE;   // Used
      osr13 : Bool := FALSE;   // Used
      osr14 : Bool := FALSE;   // Used
      osr15 : Bool := TRUE;   // Used
      osr16 : Bool := FALSE;   // Used
      osr17 : Bool := TRUE;   // Used
      osr18 : Bool := TRUE;   // Used
      osr19 : Bool := TRUE;   // Used
      osr20 : Bool := TRUE;   // Used
      osr21 : Bool := TRUE;   // Used
      osr22 : Bool := TRUE;   // Used
      osr23 : Bool := FALSE;   // Used
      osr24 : Bool := FALSE;   // Used
      osr25 : Bool := FALSE;   // Used
      osr26 : Bool := FALSE;   // Used
      osr27 : Bool := FALSE;   // Used
      osr28 : Bool := FALSE;   // Used
      osr29 : Bool := FALSE;   // Used
      osr30 : Bool := TRUE;   // Used
      osr31 : Bool := TRUE;   // Used
      osr32 : Bool := TRUE;   // Used
      osr33 : Bool := TRUE;   // Used
      osr34 : Bool := TRUE;   // Used
      osr35 : Bool := FALSE;   // Used
      osr36 : Bool := FALSE;   // Used
      osr37 : Bool := TRUE;
      osr38 : Bool := FALSE;   // Used
      osr39 : Bool := TRUE;   // Used
      osr40 : Bool := FALSE;   // Used
      osr41 : Bool := TRUE;   // Used
      osr42 : Bool := TRUE;
      osr43 : Bool := TRUE;
      osr44 : Bool := FALSE;
      osr45 : Bool := FALSE;   // Used
      osr46 : Bool := FALSE;   // Used
      osr47 : Bool := FALSE;
      osr48 : Bool := FALSE;
      osr49 : Bool := FALSE;
      osr50 : Bool := TRUE;
      osr51 : Bool := FALSE;
      osr52 : Bool := TRUE;
      osr53 : Bool := FALSE;
      osr54 : Bool := FALSE;
      osr55 : Bool := FALSE;
      osr56 : Bool := TRUE;
      osr57 : Bool := FALSE;
      osr58 : Bool := FALSE;
      osr59 : Bool := FALSE;
      osr60 : Bool := TRUE;
      osr61 : Bool := FALSE;
      osr62 : Bool := FALSE;
      osr63 : Bool := FALSE;
      osr64 : Bool := FALSE;
      osr65 : Bool := FALSE;
      osr66 : Bool := FALSE;
      osr67 : Bool := TRUE;
      osr68 : Bool := FALSE;
      osr69 : Bool := TRUE;
      osr70 : Bool := FALSE;
      osr71 : Bool := FALSE;
      osr72 : Bool := FALSE;
      osr73 : Bool := FALSE;
      osr74 : Bool := TRUE;
      osr75 : Bool := TRUE;
      osr76 : Bool := FALSE;
      osr77 : Bool := TRUE;
      osr78 : Bool := TRUE;
      osr79 : Bool := FALSE;
      osr80 : Bool := FALSE;
      osr81 : Bool := FALSE;   // Used
      osr82 : Bool := FALSE;   // Used
      osr83 : Bool := FALSE;
      osr84 : Bool := FALSE;
      osr85 : Bool := FALSE;
      osr86 : Bool := FALSE;
      osr87 : Bool := FALSE;
      osr88 : Bool := TRUE;
      osr89 : Bool := FALSE;
      osr90 : Bool := FALSE;   // Used
      osr91 : Bool := FALSE;
      osr92 : Bool := FALSE;
      osr93 : Bool := TRUE;
      osr94 : Bool := TRUE;
      osr95 : Bool := TRUE;
      osr96 : Bool := TRUE;
   END_VAR
BEGIN
END_DATA_BLOCK

DATA_BLOCK "DB03_Machine"   // DB3
{ S7_Optimized_Access := 'FALSE' }
AUTHOR : Robopac
VERSION : 0.0
// stored: AutoNumber false, IsOnlyStoredInLoadMemory false, IsWriteProtectedInAS false
   VAR RETAIN
      dbx0_0 : Bool := FALSE;   // Enable the arm rotation revolution counter
      dbx0_1 : Bool := FALSE;   // High pressure on prestretch roller dancer
      dbx0_2 : Bool := FALSE;   // One arm revolution done support memory
      dbx0_3 : Bool := FALSE;   // One arm revolution done
      dbx0_4 : Bool := FALSE;   // Support memory for revolution counter
      dbx0_5 : Bool := FALSE;   // Support memory for 10% prestretch carriage
      dbx0_6 : Bool := FALSE;
      dbx0_7 : Bool := FALSE;   // Support memory for arm rotation speed recorded
      dbb1 : Byte := 16#00;
      MachineExc : Bool := FALSE;   // Wrapping excluded
      MachineInc : Bool := FALSE;   // Wrapping included
      dbb3 : Byte := 16#00;
      dbx4_0 : Bool := FALSE;   // Memory to silent acoustic signal on alarm
      dbx4_1 : Bool := FALSE;
      dbx4_2 : Bool := FALSE;   // Condition to check all out of positon alarm
      dbx4_3 : Bool := FALSE;   // Condition for manual operation
      dbx4_4 : Bool := FALSE;   // All units are ready for automatic cycle
      dbx4_5 : Bool := FALSE;
      dbx4_6 : Bool := FALSE;   // Data for next ring height loaded
      dbx4_7 : Bool := FALSE;   // Data for next ring height loaded
      dbx5_0 : Bool := FALSE;   // Wrapping cycle: Next step is cut and pallet unload
      dbx5_1 : Bool := FALSE;   // Wrapping cycle: Next step is cut and new spool carriage height
      dbx5_2 : Bool := FALSE;   // Wrapping cycle: Next step is new spool carriage height
      dbx5_3 : Bool := FALSE;   // Wrapping cycle: After this step top waterproof
      dbx5_4 : Bool := FALSE;   // Wrong data program for the pallet on the machine
      dbx5_5 : Bool := FALSE;   // Closing upper(double) rope unit
      dbx5_6 : Bool := FALSE;   // Closing single or lower(double) rope unit
      dbx5_7 : Bool := FALSE;   // Memory for timeout enable
      dbx6_0 : Bool := FALSE;   // Memory to exclude infeed safety barrier
      dbx6_1 : Bool := FALSE;   // Memory to exclude outfeed safety barrier
      dbx6_2 : Bool := FALSE;   // Memory to exclude infeed safety barrier
      dbx6_3 : Bool := FALSE;   // Memory to exclude infeed safety barrier
      dbx6_4 : Bool := FALSE;   // Memory to exclude outfeed safety barrier
      dbx6_5 : Bool := FALSE;   // Memory to exclude outfeed safety barrier
      dbx6_6 : Bool := FALSE;
      dbx6_7 : Bool := FALSE;
      dbx7_0 : Bool := FALSE;   // Pressure plate excluded for low pallet
      dbx7_1 : Bool := FALSE;
      dbx7_2 : Bool := FALSE;   // Support memory to check rotation speed
      dbx7_3 : Bool := FALSE;   // Support memory to check spool carriage speed
      dbx7_4 : Bool := FALSE;   // Used by S7-200
      dbx7_5 : Bool := FALSE;   // Machine in wrapping cycle
      dbx7_6 : Bool := FALSE;   // Support memory to refresh pallet per hour value
      dbx7_7 : Bool := FALSE;
      dbb8 : Byte := 16#00;
      TopExc : Bool := FALSE;   // Top excluded
      TopBefore : Bool := FALSE;   // Top included before wrapping beginning
      TopWaterP : Bool := FALSE;   // Top included waterproof
      dbw10 : Int := 0;
      dbw12 : Int := 0;   // Counter for revolution on running spool carriage height
      dbw14 : Int := 0;   // Counter for revolution on welder contrast
      dbw16 : Int := 0;   // Counter for revolution of deceleration
      dbw18 : Int := 0;
      dbw20 : Int := 0;   // Active program for multiprogram (Display)
      dbw22 : Int := 0;   // Selected program for multiprogram (Display)
      dbw24 : Int := 0;   // Program to be shown on data program page (Display)
      dbw26 : Int := 0;   // Program selection by external signal
      dbw28 : Int := 0;   // Program selection by external signal
      dbw30 : Int := 0;   // Support memory for data transfer
      dbw32 : Int := 0;   // Arm rotation speed recorded (rpm*10)
      dbw34 : Int := 0;   // Required arm rotation speed recorded (%*10)
      dbw36 : Int := 0;
      dbw38 : Int := 0;   // Support memory to evaluate carriage movement speed
      dbw40 : Int := 0;   // Support memory to evaluate carriage movement speed
      dbw42 : Int := 0;   // Spool carriage movement speed mm/sec
      dbw44 : Int := 0;   // table rotation movement speed mm/sec
      dbw46 : Int := 0;   // Arm rotation speed (rpm*10) related to actual required speed
      dbw48 : Int := 0;   // Spool carriage movement speed mm/sec recorded
      dbw50 : Int := 0;
      dbw52 : Int := 0;   // High speed for spool carriage movement (%) recorded from display
      dbw54 : Int := 0;   // upport memory for spool carriage high speed
      dbw56 : Int := 0;   // Spool carriage movement speed used on cycle (mm/sec)
      dbb58 : Byte := 16#00;   // Counter for DAC M20 converter
      dbx59_0 : Bool := FALSE;   // Arm rotation and top carriage speed change for DAC M20
      dbx59_1 : Bool := FALSE;   // Spool carriage speed change for DAC M20
      dbx59_2 : Bool := FALSE;   // Counter for DAC M20 is odd
      dbx59_3 : Bool := FALSE;
      dbx59_4 : Bool := FALSE;
      dbx59_5 : Bool := FALSE;
      dbx59_6 : Bool := FALSE;
      dbx59_7 : Bool := FALSE;
      dbw60 : Int := 0;   // Value for DAC analog output
      dbw62 : Int := 0;
      dbw64 : Int := 0;
      dbw66 : Int := 0;   // Support for running height data transfer
      dbw68 : Int := 0;   // Number of the running spool carriage height
      dbw70 : Int := 0;   // Film overlap for running spool carriage height
      dbw72 : Int := 0;   // Carriage height (mm) for running spool carriage height
      dbx74_0 : Bool := FALSE;   // Landmark (0=Bottom 1=Top) for running spool carriage height
      dbx74_1 : Bool := FALSE;   // Pallet lifter for running spool carriage height (0=Excluded 1=Included)
      dbx74_2 : Bool := FALSE;   // Spare
      dbx74_3 : Bool := FALSE;   // Airblower on film tail for running spool carriage height (0=Exc 1=Inc)
      dbx74_4 : Bool := FALSE;   // Next step for running spool carriage height (0=End 1=Next)
      dbx74_5 : Bool := FALSE;   // Pressure plate for running spool carriage height (0=Excluded 1=Included)
      dbx74_6 : Bool := FALSE;   // Spare
      dbx74_7 : Bool := FALSE;   // Spare
      dbb75 : Byte := 16#00;   // Spare
      dbw76 : Int := 0;   // Revolutions for running spool carriage height
      dbb78 : Byte := 16#00;   // Rope unit for running spool carriage height (1=Excluded 2=Inc 3=Inc during)
      dbb79 : Byte := 16#00;   // Rope unit for running spool carriage height (1=Excluded 2=Inc 3=Inc during)
      dbw80 : Int := 0;   // Film force for running spool carriage height
      dbw82 : Int := 0;   // Film prestretch for running spool carriage height
      dbw84 : Int := 0;   // Delay to open or close upper rope unit for runninh spool carriage height
      dbw86 : Int := 0;   // Delay to open or close lower rope unit for runninh spool carriage height
      dbw88 : Int := 0;   // Spare for running spool carriage height
      dbw90 : Int := 0;   // Spare for running spool carriage height
      dbw92 : Int := 0;   // Spare for running spool carriage height
      dbw94 : Int := 0;   // Spare for running spool carriage height
      dbw96 : Int := 0;
      dbw98 : Int := 0;
   END_VAR
BEGIN
END_DATA_BLOCK

DATA_BLOCK "DB04_Conveyor"   // DB4
{ S7_Optimized_Access := 'FALSE' }
AUTHOR : Robopac
VERSION : 0.0
// stored: AutoNumber false, IsOnlyStoredInLoadMemory false, IsWriteProtectedInAS false
   VAR RETAIN
      dbw0 : Int := 0;
      dbw2 : Int := 0;
      dbx4_0 : Bool := TRUE;   // Pallet positioned
      dbx4_1 : Bool := FALSE;   // Deceleration for pallet positioning
      dbx4_2 : Bool := FALSE;   // Support memory for wrong pallet positioning emergency
      dbx4_3 : Bool := FALSE;   // Unload memory for outfeed conveyor
      dbx4_4 : Bool := TRUE;   // Support for end of transfer signal for pallet load/unload
      dbx4_5 : Bool := TRUE;   // Short pallet positioned
      dbx4_6 : Bool := TRUE;   // Pallet positioned for clampcutcycle
      dbx4_7 : Bool := FALSE;   // Pallet positioned from reverse
      dbb5 : Byte := 16#00;
      dbw6 : Int := 0;
      dbw8 : Int := 0;
      dbw10 : Int := 0;   // Pallet lenght measured in infeed (pulse)
      dbw12 : Int := 0;   // Pallet lenght measured in central machine (pulse)
      dbw14 : Int := 0;   // Pallet lenght measured in infeed (mm)
      dbw16 : Int := 0;   // Pallet lenght measured in central machine (mm)
      dbw18 : Int := 0;   // Half pallet lenght for selfcentering system
      dbw20 : Int := -100;   // Deceleration for pallet positioning on selfcentering system
      dbw22 : Int := 78;   // Support for conveyor movement speed
      dbw24 : Int := 0;
      dbw26 : Int := 0;
      dbw28 : Int := 0;
      dbw30 : Int := 0;
      dbw32 : Int := 0;
      dbw34 : Int := 0;
      dbd36 : DInt := 0;
      dbd40 : DInt := 0;
      dbd44 : DInt := 0;
      dbd48 : DInt := 0;
      dbd52 : DInt := 0;
      dbd56 : DInt := 0;
      dbd60 : DInt := 0;
      dbd64 : DInt := 0;
      dbd68 : DInt := 0;
      dbd72 : DInt := 0;
      dbw76 : Int := 0;
      dbb78 : Byte := 16#00;   // Rope unit for running spool carriage height (1=Excluded 2=Inc 3=Inc during
      dbb79 : Byte := 16#00;   // Rope unit for running spool carriage height (1=Excluded 2=Inc 3=Inc during
      dbd80 : DInt := 0;
      dbd84 : DInt := 0;
   END_VAR
BEGIN
END_DATA_BLOCK

DATA_BLOCK "DB05_SpoolCarriagePos"   // DB5
{ S7_Optimized_Access := 'FALSE' }
AUTHOR : Robopac
VERSION : 0.0
// stored: AutoNumber false, IsOnlyStoredInLoadMemory false, IsWriteProtectedInAS false
   VAR RETAIN
      dbx0_0 : Bool := FALSE;   // Table rotation forward
      dbx0_1 : Bool := FALSE;   // Table rotation backward
      dbx0_2 : Bool := FALSE;   // Table rotation speed: Low
      dbx0_3 : Bool := FALSE;   // Table rotation speed: Middle 1 for top
      dbx0_4 : Bool := FALSE;   // Table rotation speed: Middle 2 for welder contrast
      dbx0_5 : Bool := FALSE;   // Table rotation speed: High
      dbx0_6 : Bool := FALSE;
      dbx0_7 : Bool := FALSE;
      dbx1_0 : Bool := FALSE;   // Spool carriage axis movement upward
      dbx1_1 : Bool := FALSE;   // Spool carriage axis movement downward
      dbx1_2 : Bool := FALSE;   // Spool carriage axis movement inside low speed area
      dbx1_3 : Bool := FALSE;   // Spool carriage axis movement low speed
      dbx1_4 : Bool := FALSE;   // Spool carriage upward
      dbx1_5 : Bool := FALSE;   // Spool carriage downward
      dbx1_6 : Bool := FALSE;
      dbx1_7 : Bool := FALSE;
      dbx2_0 : Bool := FALSE;
      dbx2_1 : Bool := FALSE;   // Support memory for enable (EN) on table rotation and table conveyor inverter
      dbx2_2 : Bool := FALSE;
      dbx2_3 : Bool := FALSE;
      dbx2_4 : Bool := FALSE;
      dbx2_5 : Bool := FALSE;
      dbx2_6 : Bool := FALSE;
      dbx2_7 : Bool := FALSE;
      dbx3_0 : Bool := FALSE;   // Spool carriage: Support for encoder running control
      dbx3_1 : Bool := FALSE;   // Spool carriage: Support for encoder running control alarm
      dbx3_2 : Bool := FALSE;
      dbx3_3 : Bool := FALSE;
      dbx3_4 : Bool := FALSE;
      dbx3_5 : Bool := FALSE;
      dbx3_6 : Bool := FALSE;
      dbx3_7 : Bool := FALSE;
      dbx4_0 : Bool := FALSE;   // Pallet height recording in automatic mode
      dbx4_1 : Bool := FALSE;   // Support memory for pallet height recording
      dbx4_2 : Bool := FALSE;
      dbx4_3 : Bool := FALSE;   // Support memory for pallet height filter
      dbx4_4 : Bool := FALSE;   // Condition for pallet height detected
      dbx4_5 : Bool := FALSE;
      dbx4_6 : Bool := TRUE;   // Carriage in position to rotate in medium to wrap top
      dbx4_7 : Bool := FALSE;
      dbx5_0 : Bool := FALSE;
      dbx5_1 : Bool := FALSE;
      dbx5_2 : Bool := FALSE;
      dbx5_3 : Bool := FALSE;
      dbx5_4 : Bool := TRUE;   // Top wrapped ring position
      dbw6 : Int := 100;   // Spool carriage: Support for movement speed
      dbw8 : Int := 50;   // Spool carriage: Support for movement deceleration
      dbw10 : Int := 100;
      dbw12 : Int := 10199;
      dbw14 : Int := 10306;   // Pallet height on machine conveyor + 300 mm
      dbw16 : Int := 9999;   // Pallet height on machine conveyor
      dbw18 : Int := 9999;   // Pallet height on machine conveyor
      dbw20 : Int := 480;   // Spool carriage height for middle speed on welder contrast
      dbw22 : Int := -2;   // Support memory for pallet height filter
      dbw24 : Int := 0;   // Support memory for pallet height
      dbw26 : Int := -380;   // Spool carriage height for middle speed before top cycle
      dbw28 : Int := 0;
      dbd30 : DInt := -1;   // Spool carriage position: Pulse
      dbw34 : Int := -2;   // Spool carriage position: Top of the spool
      dbw36 : Int := 1782;   // Spool carriage position: Spool carriage all up position
      dbw38 : Int := 50;   // Spool carriage position: Deceleration position for carriage overrun down
      dbw40 : Int := 1732;   // Spool carriage position: Deceleration position for carriage overrun up
      dbd42 : DInt := -1;   // Support for encoder spool carriage running control
      dbw46 : Int := 12;   // Support for encoder spool carriage running control
      dbw48 : Int := 0;
      dbw50 : Int := 0;   // Support memory for machine conveyor speed (%)
      dbw52 : Int := 0;   // Support memory for spool carriage and machine conveyor speed (%)
      dbw54 : Int := 0;   // Support memory for for arm rotation speed (%*10)
      dbw56 : Int := 0;   // Support memory for top carriage forward/backward speed (%*10)
      dbw58 : Int := 0;   // Support memory for top carriage forward/backward and arm rotation speed (%*10)
      dbw60 : Int := 0;
      dbw62 : Int := 0;
      dbw64 : Int := 0;
      dbw66 : Int := 0;
      dbw68 : Int := 0;
      Req1_Start : Bool := FALSE;   // Positioning request 1: Start
      Req2_Start : Bool := FALSE;   // Positioning request 2: Start
      Req3_Start : Bool := FALSE;   // Positioning request 3: Start
      Req4_Start : Bool := FALSE;   // Positioning request 4: Start
      Req5_Start : Bool := FALSE;   // Positioning request 5: Start
      Req6_Start : Bool := FALSE;   // Positioning request 6: Start
      Req7_Start : Bool := FALSE;   // Positioning request 7: Start
      Req8_Start : Bool := FALSE;   // Positioning request 8: Start
      Req9_Start : Bool := FALSE;   // Positioning request 9: Start
      Req10_Start : Bool := FALSE;   // Positioning request 10: Start
      Req1_Dest : Int := 50;   // Positioning request 1: Destination position
      Req2_Dest : Int := 40;   // Positioning request 2: Destination position
      Req3_Dest : Int := -260;   // Positioning request 3: Destination position
      Req4_Dest : Int := 0;   // Positioning request 4: Destination position
      Req1_Fwd : Bool := FALSE;   // Positioning request 1: Axis forward
      Req1_Bkw : Bool := FALSE;   // Positioning request 1: Axis backward
      Req1_Slow : Bool := FALSE;   // Positioning request 1: Axis slow speed
      Req1_Pos : Bool := FALSE;   // Positioning request 1: Axis in position
      Req2_Fwd : Bool := FALSE;   // Positioning request 2: Axis forward
      Req2_Bkw : Bool := FALSE;   // Positioning request 2: Axis backward
      Req2_Slow : Bool := FALSE;   // Positioning request 2: Axis slow speed
      Req2_Pos : Bool := FALSE;   // Positioning request 2: Axis in position
      Req3_Fwd : Bool := FALSE;   // Positioning request 3: Axis forward
      Req3_Bkw : Bool := FALSE;   // Positioning request 3: Axis backward
      Req3_Slow : Bool := FALSE;   // Positioning request 3: Axis slow speed
      Req3_Pos : Bool := FALSE;   // Positioning request 3: Axis in position
      Req4_Fwd : Bool := FALSE;   // Positioning request 4: Axis forward
      Req4_Bkw : Bool := FALSE;   // Positioning request 4: Axis backward
      Req4_Slow : Bool := FALSE;   // Positioning request 4: Axis slow speed
      Req4_Pos : Bool := FALSE;   // Positioning request 4: Axis in position
      Req5_Dest : Int := 0;   // Positioning request 5: Destination position
      Req6_Dest : Int := 0;   // Positioning request 6: Destination position
      Req7_Dest : Int := 0;   // Positioning request 7: Destination position
      Req8_Dest : Int := 0;   // Positioning request 8: Destination position
      Req5_Fwd : Bool := FALSE;   // Positioning request 5: Axis forward
      Req5_Bkw : Bool := FALSE;   // Positioning request 5: Axis backward
      Req5_Slow : Bool := FALSE;   // Positioning request 5: Axis slow speed
      Req5_Pos : Bool := FALSE;   // Positioning request 5: Axis in position
      Req6_Fwd : Bool := FALSE;   // Positioning request 6: Axis forward
      Req6_Bkw : Bool := FALSE;   // Positioning request 6: Axis backward
      Req6_Slow : Bool := FALSE;   // Positioning request 6: Axis slow speed
      Req6_Pos : Bool := FALSE;   // Positioning request 6: Axis in position
      Req7_Fwd : Bool := FALSE;   // Positioning request 7: Axis forward
      Req7_Bkw : Bool := FALSE;   // Positioning request 7: Axis backward
      Req7_Slow : Bool := FALSE;   // Positioning request 7: Axis slow speed
      Req7_Pos : Bool := FALSE;   // Positioning request 7: Axis in position
      Req8_Fwd : Bool := FALSE;   // Positioning request 8: Axis forward
      Req8_Bkw : Bool := FALSE;   // Positioning request 8: Axis backward
      Req8_Slow : Bool := FALSE;   // Positioning request 8: Axis slow speed
      Req8_Pos : Bool := FALSE;   // Positioning request 8: Axis in position
      dbw92 : Int := 2000;   // Time for arm rotation motor stop
      dbw94 : Int := 0;
      dbw96 : Int := 0;
      dbw98 : Int := 0;   // Time for conveyor motor stop
      dbw100 : Int := 0;   // Time for forward on arm rotation and conveyor inverter
      dbw102 : Int := 0;   // Time for backward on arm rotation and conveyor inverter
      dbw104 : Int := 0;
      dbw106 : Int := 0;
      dbw108 : Int := 0;
      dbw110 : Int := 0;
   END_VAR
BEGIN
END_DATA_BLOCK

DATA_BLOCK "DB06_Clamp"   // DB6
{ S7_Optimized_Access := 'FALSE' }
AUTHOR : Robopac
VERSION : 0.0
// stored: AutoNumber false, IsOnlyStoredInLoadMemory false, IsWriteProtectedInAS false
   VAR RETAIN
      dbx0_0 : Bool := FALSE;   // Welder contrast upward
      dbx0_1 : Bool := FALSE;   // Welder contrast downward
      dbx0_2 : Bool := FALSE;   // Welder unit upward
      dbx0_3 : Bool := FALSE;   // Welder unit downward
      dbx0_4 : Bool := FALSE;
      dbx0_5 : Bool := FALSE;   // Film clamp upward
      dbx0_6 : Bool := FALSE;   // Film clamp downward
      dbx0_7 : Bool := FALSE;   // Welder and cut unit forward
      dbx1_0 : Bool := FALSE;   // Welder and cut unit backward
      dbx1_1 : Bool := FALSE;
      dbx1_2 : Bool := FALSE;
      dbx1_3 : Bool := FALSE;
      dbx1_4 : Bool := FALSE;
      dbx1_5 : Bool := FALSE;
      dbx1_6 : Bool := FALSE;
      dbx1_7 : Bool := FALSE;
      dbx2_0 : Bool := FALSE;   // Welder contrast forward
      dbx2_1 : Bool := FALSE;   // Welder contrast backward
      dbx2_2 : Bool := FALSE;
      dbx2_3 : Bool := FALSE;
      dbx2_4 : Bool := FALSE;
      dbx2_5 : Bool := FALSE;
      dbx2_6 : Bool := FALSE;
      dbx2_7 : Bool := FALSE;
      dbb3 : Byte := 16#00;
      dbx4_0 : Bool := FALSE;   // Spool carrage upward to cover tail
      dbx4_1 : Bool := FALSE;   // Spool carrage downward after film tail covered
      dbx4_2 : Bool := FALSE;   // Spool carrage upward at the begining
      dbx4_3 : Bool := FALSE;   // Spool carriage height to pull film at begining
      dbx4_4 : Bool := FALSE;   // Support memory for revolution over welder contrast
      dbx4_5 : Bool := TRUE;   // Clamp carriage is not backward because wrapping cycle
      dbb5 : Byte := 16#00;
      dbw6 : Int := 0;
      dbw8 : Int := 0;
      dbw10 : Int := 500;   // Spool carriage height for film tail airblower
      dbw12 : Int := 0;   // Number of revolution to open clamp
      dbw14 : Int := 0;   // Spool carriage height for film tail wrapped
      dbw16 : Int := 200;   // Spool carriage height to enable revolution over clamp
      dbw18 : Int := 1942;
      dbw20 : Int := 0;
      dbw22 : Int := 0;
      dbw24 : Int := 0;
      dbw26 : Int := 0;
      dbw28 : Int := 0;
      dbw30 : Int := 0;
      dbw32 : Int := 0;
      dbw34 : Int := 0;
      dbw36 : Int := 0;
      dbw38 : Int := 0;
      dbw40 : Int := 0;   // Delay to open clamp (number of 100msec)
      dbw42 : Int := 0;   // Time to open clamp related to actual speed
      dbw44 : Int := 0;
      dbw46 : Int := 0;
      dbw48 : Int := 0;
   END_VAR
BEGIN
END_DATA_BLOCK

DATA_BLOCK "DB07_TopAux"   // DB7
{ S7_Optimized_Access := 'FALSE' }
AUTHOR : Robopac
VERSION : 0.0
// stored: AutoNumber false, IsOnlyStoredInLoadMemory false, IsWriteProtectedInAS false
   VAR RETAIN
      VB700 : Byte := 16#00;
      V701_0 : Bool := TRUE;   // Top film is wrapped
      V701_1 : Bool := FALSE;   // Support memory for top wrapped
      V701_2 : Bool := FALSE;
      V701_3 : Bool := FALSE;
      V701_4 : Bool := FALSE;
      V701_5 : Bool := FALSE;
      V701_6 : Bool := FALSE;
      V701_7 : Bool := FALSE;
   END_VAR
BEGIN
END_DATA_BLOCK

DATA_BLOCK "DB08_Prestretch"   // DB8
{ S7_Optimized_Access := 'FALSE' }
AUTHOR : Robopac
VERSION : 0.0
// stored: AutoNumber false, IsOnlyStoredInLoadMemory false, IsWriteProtectedInAS false
   VAR RETAIN
      dbx0_0 : Bool := FALSE;   // Support memory for prestretch PGSM or PGSA
      dbx0_1 : Bool := FALSE;
      dbx0_2 : Bool := FALSE;
      dbx0_3 : Bool := FALSE;
      dbx0_4 : Bool := FALSE;
      dbx0_5 : Bool := FALSE;
      dbx0_6 : Bool := FALSE;
      dbx0_7 : Bool := FALSE;
      dbw2 : Int := 0;
      dbw4 : Int := 0;
      dbw6 : Int := 0;
      dbw8 : Int := 0;
      dbw10 : Int := 0;   // Film provided for every revolution at max speed (mm per revolution)
      dbw12 : Int := 0;   // Film force value to apply to pallet (mm)
      dbd14 : DInt := 0;   // Support memory for film force to apply to pallet
      dbw18 : Int := 0;   // Film force value to apply to pallet (analog value)
      dbw20 : Int := 0;   // Film force value to apply to pallet (%)
      dbw22 : Int := 0;
      dbw24 : Int := 0;
      dbw26 : Int := 0;
      dbw28 : Int := 0;
      dbw30 : Int := 0;   // Gain for analog scaling
      dbw32 : Int := 200;   // Film prestretch value to apply to pallet
      dbd34 : DInt := 0;   // Support memory for film prestretch to apply to pallet
      dbw38 : Int := 102;   // Film prestretch value to apply to pallet (analog value)
      dbw40 : Int := 0;
      dbw42 : Int := 0;
      dbw44 : Int := 0;
      dbw46 : Int := 0;
      dbw48 : Int := 0;
      dbw50 : Int := 0;   // Support for film prestretch test
      dbw52 : Int := 0;   // Support for film prestretch test
      dbw54 : Int := 0;   // Film weight every mm of film (10^-5 g/mm)
      dbw56 : Int := 0;
      dbw58 : Int := 0;
      dbw60 : Int := 0;
   END_VAR
BEGIN
END_DATA_BLOCK

